gfCNCPoint1[6054] = {X 351.3681, Y 35.6206, Z -1.3333, A 0.000, B 0.000, C 0.000 }
gfCNCPoint1[6055] = {X 352.4747, Y 34.8217, Z -1.3333, A 0.000, B 0.000, C 0.000 }
gfCNCPoint1[6056] = {X 353.5730, Y 33.7520, Z -1.3333, A 0.000, B 0.000, C 0.000 }
gfCNCPoint1[6057] = {X 354.5237, Y 32.5493, Z -1.3333, A 0.000, B 0.000, C 0.000 }
gfCNCPoint1[6058] = {X 355.3108, Y 31.2336, Z -1.3333, A 0.000, B 0.000, C 0.000 }
gfCNCPoint1[6059] = {X 355.9209, Y 29.8271, Z -1.3333, A 0.000, B 0.000, C 0.000 }
gfCNCPoint1[6060] = {X 356.3440, Y 28.3535, Z -1.3333, A 0.000, B 0.000, C 0.000 }
gfCNCPoint1[6061] = {X 356.6085, Y 26.7184, Z -1.3333, A 0.000, B 0.000, C 0.000 }
gfCNCPoint1[6062] = {X 356.7162, Y 25.0656, Z -1.3333, A 0.000, B 0.000, C 0.000 }
gfCNCPoint1[6063] = {X 356.6661, Y 23.4100, Z -1.3333, A 0.000, B 0.000, C 0.000 }
gfCNCPoint1[6064] = {X 356.4586, Y 21.7667, Z -1.3333, A 0.000, B 0.000, C 0.000 }
gfCNCPoint1[6065] = {X 356.1382, Y 20.3836, Z -1.3333, A 0.000, B 0.000, C 0.000 }
gfCNCPoint1[6066] = {X 355.6490, Y 19.0509, Z -1.3333, A 0.000, B 0.000, C 0.000 }
gfCNCPoint1[6067] = {X 354.9985, Y 17.7891, Z -1.3333, A 0.000, B 0.000, C 0.000 }
gfCNCPoint1[6068] = {X 354.1969, Y 16.6174, Z -1.3333, A 0.000, B 0.000, C 0.000 }
gfCNCPoint1[6069] = {X 353.3646, Y 15.6889, Z -1.3333, A 0.000, B 0.000, C 0.000 }
gfCNCPoint1[6070] = {X 352.4079, Y 14.8891, Z -1.3333, A 0.000, B 0.000, C 0.000 }
gfCNCPoint1[6071] = {X 351.3465, Y 14.2346, Z -1.3333, A 0.000, B 0.000, C 0.000 }
gfCNCPoint1[6072] = {X 350.2023, Y 13.7390, Z -1.3333, A 0.000, B 0.000, C 0.000 }
gfCNCPoint1[6073] = {X 348.9989, Y 13.4124, Z -1.3333, A 0.000, B 0.000, C 0.000 }
gfCNCPoint1[6074] = {X 347.3616, Y 13.2058, Z -1.3333, A 0.000, B 0.000, C 0.000 }
gfCNCPoint1[6075] = {X 345.7114, Y 13.2112, Z -1.3333, A 0.000, B 0.000, C 0.000 }
gfCNCPoint1[6076] = {X 344.0755, Y 13.4284, Z -1.3333, A 0.000, B 0.000, C 0.000 }
gfCNCPoint1[6077] = {X 342.4811, Y 13.8538, Z -1.3333, A 0.000, B 0.000, C 0.000 }
gfCNCPoint1[6078] = {X 340.9545, Y 14.4805, Z -1.3333, A 0.000, B 0.000, C 0.000 }
gfCNCPoint1[6079] = {X 339.5210, Y 15.2981, Z -1.3333, A 0.000, B 0.000, C 0.000 }
gfCNCPoint1[6080] = {X 339.4274, Y 16.1841, Z -1.3333, A 0.000, B 0.000, C 0.000 }
gfCNCPoint1[6081] = {X 339.1743, Y 17.0384, Z -1.3333, A 0.000, B 0.000, C 0.000 }
gfCNCPoint1[6082] = {X 338.7701, Y 17.8324, Z -1.3333, A 0.000, B 0.000, C 0.000 }
gfCNCPoint1[6083] = {X 338.2283, Y 18.5396, Z -1.3333, A 0.000, B 0.000, C 0.000 }
gfCNCPoint1[6084] = {X 337.5670, Y 19.1366, Z -1.3333, A 0.000, B 0.000, C 0.000 }
gfCNCPoint1[6085] = {X 336.8399, Y 19.6716, Z -1.3333, A 0.000, B 0.000, C 0.000 }
gfCNCPoint1[6086] = {X 335.9170, Y 20.1909, Z -1.3333, A 0.000, B 0.000, C 0.000 }
gfCNCPoint1[6087] = {X 334.9039, Y 20.4988, Z -1.3333, A 0.000, B 0.000, C 0.000 }
gfCNCPoint1[6088] = {X 333.8481, Y 20.5809, Z -1.3333, A 0.000, B 0.000, C 0.000 }
gfCNCPoint1[6089] = {X 332.7995, Y 20.4334, Z -1.3333, A 0.000, B 0.000, C 0.000 }
gfCNCPoint1[6090] = {X 331.8074, Y 20.0631, Z -1.3333, A 0.000, B 0.000, C 0.000 }
gfCNCPoint1[6091] = {X 330.9185, Y 19.4875, Z -1.3333, A 0.000, B 0.000, C 0.000 }
gfCNCPoint1[6092] = {X 330.1748, Y 18.7338, Z -1.3333, A 0.000, B 0.000, C 0.000 }
gfCNCPoint1[6093] = {X 329.6111, Y 17.8373, Z -1.3333, A 0.000, B 0.000, C 0.000 }
gfCNCPoint1[6094] = {X 326.0906, Y 10.5950, Z -1.3333, A 0.000, B 0.000, C 0.000 }
gfCNCPoint1[6095] = {X 325.7555, Y 9.6856, Z -1.3333, A 0.000, B 0.000, C 0.000 }
gfCNCPoint1[6096] = {X 325.6068, Y 8.7279, Z -1.3333, A 0.000, B 0.000, C 0.000 }
gfCNCPoint1[6097] = {X 325.6502, Y 7.7597, Z -1.3333, A 0.000, B 0.000, C 0.000 }
gfCNCPoint1[6098] = {X 325.8841, Y 6.8192, Z -1.3333, A 0.000, B 0.000, C 0.000 }
gfCNCPoint1[6099] = {X 326.2993, Y 5.9435, Z -1.3333, A 0.000, B 0.000, C 0.000 }
gfCNCPoint1[6100] = {X 326.9295, Y 5.1131, Z -1.3333, A 0.000, B 0.000, C 0.000 }
gfCNCPoint1[6101] = {X 327.7216, Y 4.4356, Z -1.3333, A 0.000, B 0.000, C 0.000 }
gfCNCPoint1[6102] = {X 328.3967, Y 3.9733, Z -1.3333, A 0.000, B 0.000, C 0.000 }
gfCNCPoint1[6103] = {X 329.3298, Y 3.4827, Z -1.3333, A 0.000, B 0.000, C 0.000 }
gfCNCPoint1[6104] = {X 330.3464, Y 3.2039, Z -1.3333, A 0.000, B 0.000, C 0.000 }
gfCNCPoint1[6105] = {X 331.3992, Y 3.1499, Z -1.3333, A 0.000, B 0.000, C 0.000 }
gfCNCPoint1[6106] = {X 332.4390, Y 3.3233, Z -1.3333, A 0.000, B 0.000, C 0.000 }
gfCNCPoint1[6107] = {X 333.3767, Y 2.7966, Z -1.3333, A 0.000, B 0.000, C 0.000 }
gfCNCPoint1[6108] = {X 334.3334, Y 2.3051, Z -1.3333, A 0.000, B 0.000, C 0.000 }
gfCNCPoint1[6109] = {X 334.5448, Y 2.7361, Z -1.3333, A 0.000, B 0.000, C 0.000 }
gfCNCPoint1[6110] = {X 335.0204, Y 2.5083, Z -1.3333, A 0.000, B 0.000, C 0.000 }
gfCNCPoint1[6111] = {X 335.5002, Y 2.2893, Z -1.3333, A 0.000, B 0.000, C 0.000 }
gfCNCPoint1[6112] = {X 335.8480, Y 2.1345, Z -1.3333, A 0.000, B 0.000, C 0.000 }
gfCNCPoint1[6113] = {X 337.9511, Y 1.3140, Z -1.3333, A 0.000, B 0.000, C 0.000 }
gfCNCPoint1[6114] = {X 340.1167, Y 0.6764, Z -1.3333, A 0.000, B 0.000, C 0.000 }
gfCNCPoint1[6115] = {X 342.3290, Y 0.2265, Z -1.3333, A 0.000, B 0.000, C 0.000 }
gfCNCPoint1[6116] = {X 344.5716, Y -0.0325, Z -1.3333, A 0.000, B 0.000, C 0.000 }
gfCNCPoint1[6117] = {X 346.8281, Y -0.0986, Z -1.3333, A 0.000, B 0.000, C 0.000 }
gfCNCPoint1[6118] = {X 349.0821, Y 0.0286, Z -1.3333, A 0.000, B 0.000, C 0.000 }
gfCNCPoint1[6119] = {X 351.3169, Y 0.3481, Z -1.3333, A 0.000, B 0.000, C 0.000 }
gfCNCPoint1[6120] = {X 351.8868, Y 0.4533, Z -1.3333, A 0.000, B 0.000, C 0.000 }
gfCNCPoint1[6121] = {X 353.8281, Y 0.9413, Z -1.3333, A 0.000, B 0.000, C 0.000 }
gfCNCPoint1[6122] = {X 355.7145, Y 1.6111, Z -1.3333, A 0.000, B 0.000, C 0.000 }
gfCNCPoint1[6123] = {X 357.5290, Y 2.4565, Z -1.3333, A 0.000, B 0.000, C 0.000 }
gfCNCPoint1[6124] = {X 359.2553, Y 3.4699, Z -1.3333, A 0.000, B 0.000, C 0.000 }
gfCNCPoint1[6125] = {X 360.8778, Y 4.6423, Z -1.3333, A 0.000, B 0.000, C 0.000 }
gfCNCPoint1[6126] = {X 362.3820, Y 5.9632, Z -1.3333, A 0.000, B 0.000, C 0.000 }
gfCNCPoint1[6127] = {X 363.7542, Y 7.4205, Z -1.3333, A 0.000, B 0.000, C 0.000 }
gfCNCPoint1[6128] = {X 365.2289, Y 9.3236, Z -1.3333, A 0.000, B 0.000, C 0.000 }
gfCNCPoint1[6129] = {X 366.5120, Y 11.3606, Z -1.3333, A 0.000, B 0.000, C 0.000 }
gfCNCPoint1[6130] = {X 367.5917, Y 13.5125, Z -1.3333, A 0.000, B 0.000, C 0.000 }
gfCNCPoint1[6131] = {X 368.4575, Y 15.7589, Z -1.3333, A 0.000, B 0.000, C 0.000 }
gfCNCPoint1[6132] = {X 369.1015, Y 18.0787, Z -1.3333, A 0.000, B 0.000, C 0.000 }
gfCNCPoint1[6133] = {X 369.5814, Y 20.7163, Z -1.3333, A 0.000, B 0.000, C 0.000 }
gfCNCPoint1[6134] = {X 369.8368, Y 23.3851, Z -1.3333, A 0.000, B 0.000, C 0.000 }
gfCNCPoint1[6135] = {X 369.8659, Y 26.0659, Z -1.3333, A 0.000, B 0.000, C 0.000 }
gfCNCPoint1[6136] = {X 369.6685, Y 28.7395, Z -1.3333, A 0.000, B 0.000, C 0.000 }
gfCNCPoint1[6137] = {X 369.2461, Y 31.3870, Z -1.3333, A 0.000, B 0.000, C 0.000 }
gfCNCPoint1[6138] = {X 368.7206, Y 33.4984, Z -1.3333, A 0.000, B 0.000, C 0.000 }
gfCNCPoint1[6139] = {X 368.0105, Y 35.5551, Z -1.3333, A 0.000, B 0.000, C 0.000 }
gfCNCPoint1[6140] = {X 367.1214, Y 37.5409, Z -1.3333, A 0.000, B 0.000, C 0.000 }
gfCNCPoint1[6141] = {X 366.0603, Y 39.4405, Z -1.3333, A 0.000, B 0.000, C 0.000 }
gfCNCPoint1[6142] = {X 364.8354, Y 41.2387, Z -1.3333, A 0.000, B 0.000, C 0.000 }
gfCNCPoint1[6143] = {X 363.6033, Y 42.7570, Z -1.3333, A 0.000, B 0.000, C 0.000 }
gfCNCPoint1[6144] = {X 362.2428, Y 44.1612, Z -1.3333, A 0.000, B 0.000, C 0.000 }
gfCNCPoint1[6145] = {X 360.7642, Y 45.4407, Z -1.3333, A 0.000, B 0.000, C 0.000 }
gfCNCPoint1[6146] = {X 359.1791, Y 46.5854, Z -1.3333, A 0.000, B 0.000, C 0.000 }
gfCNCPoint1[6147] = {X 357.4997, Y 47.5867, Z -1.3333, A 0.000, B 0.000, C 0.000 }
gfCNCPoint1[6148] = {X 355.5329, Y 48.4795, Z -1.3333, A 0.000, B 0.000, C 0.000 }
gfCNCPoint1[6149] = {X 353.4902, Y 49.1814, Z -1.3333, A 0.000, B 0.000, C 0.000 }
gfCNCPoint1[6150] = {X 351.3901, Y 49.6861, Z -1.3333, A 0.000, B 0.000, C 0.000 }
gfCNCPoint1[6151] = {X 349.2515, Y 49.9891, Z -1.3333, A 0.000, B 0.000, C 0.000 }
gfCNCPoint1[6152] = {X 347.0938, Y 50.0876, Z -1.3333, A 0.000, B 0.000, C 0.000 }
gfCNCPoint1[6153] = {X 345.0197, Y 50.0525, Z -1.3333, A 0.000, B 0.000, C 0.000 }
gfCNCPoint1[6154] = {X 342.9564, Y 49.8375, Z -1.3333, A 0.000, B 0.000, C 0.000 }
gfCNCPoint1[6155] = {X 340.9196, Y 49.4444, Z -1.3333, A 0.000, B 0.000, C 0.000 }
gfCNCPoint1[6156] = {X 338.9245, Y 48.8760, Z -1.3333, A 0.000, B 0.000, C 0.000 }
gfCNCPoint1[6157] = {X 336.9863, Y 48.1366, Z -1.3333, A 0.000, B 0.000, C 0.000 }
gfCNCPoint1[6158] = {X 335.1196, Y 47.2319, Z -1.3333, A 0.000, B 0.000, C 0.000 }
gfCNCPoint1[6159] = {X 333.5425, Y 46.2572, Z -1.3333, A 0.000, B 0.000, C 0.000 }
gfCNCPoint1[6160] = {X 332.0447, Y 45.1645, Z -1.3333, A 0.000, B 0.000, C 0.000 }
gfCNCPoint1[6161] = {X 330.6350, Y 43.9603, Z -1.3333, A 0.000, B 0.000, C 0.000 }
gfCNCPoint1[6162] = {X 329.6763, Y 43.9518, Z -1.3333, A 0.000, B 0.000, C 0.000 }
gfCNCPoint1[6163] = {X 328.7422, Y 43.7359, Z -1.3333, A 0.000, B 0.000, C 0.000 }
gfCNCPoint1[6164] = {X 327.8771, Y 43.3228, Z -1.3333, A 0.000, B 0.000, C 0.000 }
gfCNCPoint1[6165] = {X 327.1219, Y 42.7321, Z -1.3333, A 0.000, B 0.000, C 0.000 }
gfCNCPoint1[6166] = {X 326.5249, Y 42.1498, Z -1.3333, A 0.000, B 0.000, C 0.000 }
gfCNCPoint1[6167] = {X 325.8848, Y 41.3619, Z -1.3333, A 0.000, B 0.000, C 0.000 }
gfCNCPoint1[6168] = {X 325.4424, Y 40.4483, Z -1.3333, A 0.000, B 0.000, C 0.000 }
gfCNCPoint1[6169] = {X 325.2210, Y 39.4576, Z -1.3333, A 0.000, B 0.000, C 0.000 }
gfCNCPoint1[6170] = {X 325.2326, Y 38.4426, Z -1.3333, A 0.000, B 0.000, C 0.000 }
gfCNCPoint1[6171] = {X 325.4765, Y 37.4572, Z -1.3333, A 0.000, B 0.000, C 0.000 }
gfCNCPoint1[6172] = {X 325.9397, Y 36.5539, Z -1.3333, A 0.000, B 0.000, C 0.000 }
gfCNCPoint1[6173] = {X 330.1988, Y 30.1861, Z -1.3333, A 0.000, B 0.000, C 0.000 }
gfCNCPoint1[6174] = {X 330.8195, Y 29.4619, Z -1.3333, A 0.000, B 0.000, C 0.000 }
gfCNCPoint1[6175] = {X 331.5817, Y 28.8884, Z -1.3333, A 0.000, B 0.000, C 0.000 }
gfCNCPoint1[6176] = {X 332.4495, Y 28.4927, Z -1.3333, A 0.000, B 0.000, C 0.000 }
gfCNCPoint1[6177] = {X 333.3822, Y 28.2932, Z -1.3333, A 0.000, B 0.000, C 0.000 }
gfCNCPoint1[6178] = {X 334.3360, Y 28.2995, Z -1.3333, A 0.000, B 0.000, C 0.000 }
gfCNCPoint1[6179] = {X 335.2660, Y 28.5111, Z -1.3333, A 0.000, B 0.000, C 0.000 }
gfCNCPoint1[6180] = {X 336.1286, Y 28.9182, Z -1.3333, A 0.000, B 0.000, C 0.000 }
gfCNCPoint1[6181] = {X 336.8832, Y 29.5016, Z -1.3333, A 0.000, B 0.000, C 0.000 }
gfCNCPoint1[6182] = {X 337.4845, Y 30.0811, Z -1.3333, A 0.000, B 0.000, C 0.000 }
gfCNCPoint1[6183] = {X 338.1274, Y 30.8804, Z -1.3333, A 0.000, B 0.000, C 0.000 }
gfCNCPoint1[6184] = {X 338.5678, Y 31.8068, Z -1.3333, A 0.000, B 0.000, C 0.000 }
gfCNCPoint1[6185] = {X 338.7817, Y 32.8100, Z -1.3333, A 0.000, B 0.000, C 0.000 }
gfCNCPoint1[6186] = {X 338.7575, Y 33.8355, Z -1.3333, A 0.000, B 0.000, C 0.000 }
gfCNCPoint1[6187] = {X 339.5029, Y 34.5092, Z -1.3333, A 0.000, B 0.000, C 0.000 }
gfCNCPoint1[6188] = {X 340.2812, Y 35.1446, Z -1.3333, A 0.000, B 0.000, C 0.000 }
gfCNCPoint1[6189] = {X 341.4925, Y 35.9471, Z -1.3333, A 0.000, B 0.000, C 0.000 }
gfCNCPoint1[6190] = {X 342.8028, Y 36.5754, Z -1.3333, A 0.000, B 0.000, C 0.000 }
gfCNCPoint1[6191] = {X 344.1871, Y 37.0173, Z -1.3333, A 0.000, B 0.000, C 0.000 }
gfCNCPoint1[6192] = {X 345.6190, Y 37.2646, Z -1.3333, A 0.000, B 0.000, C 0.000 }
gfCNCPoint1[6193] = {X 347.0713, Y 37.3125, Z -1.3333, A 0.000, B 0.000, C 0.000 }
gfCNCPoint1[6194] = {X 347.5133, Y 37.2896, Z -1.3333, A 0.000, B 0.000, C 0.000 }
gfCNCPoint1[6195] = {X 348.9438, Y 37.0973, Z -1.3333, A 0.000, B 0.000, C 0.000 }
gfCNCPoint1[6196] = {X 350.3238, Y 36.6741, Z -1.3333, A 0.000, B 0.000, C 0.000 }
gfCNCPoint1[6197] = {X 351.6163, Y 36.0314, Z -1.3333, A 0.000, B 0.000, C 0.000 }
gfCNCPoint1[6198] = {X 352.7866, Y 35.1865, Z -1.3333, A 0.000, B 0.000, C 0.000 }
gfCNCPoint1[6199] = {X 353.9297, Y 34.0732, Z -1.3333, A 0.000, B 0.000, C 0.000 }
gfCNCPoint1[6200] = {X 354.9191, Y 32.8214, Z -1.3333, A 0.000, B 0.000, C 0.000 }
gfCNCPoint1[6201] = {X 355.7382, Y 31.4519, Z -1.3333, A 0.000, B 0.000, C 0.000 }
gfCNCPoint1[6202] = {X 356.3731, Y 29.9880, Z -1.3333, A 0.000, B 0.000, C 0.000 }
gfCNCPoint1[6203] = {X 356.8133, Y 28.4543, Z -1.3333, A 0.000, B 0.000, C 0.000 }
gfCNCPoint1[6204] = {X 357.0854, Y 26.7729, Z -1.3333, A 0.000, B 0.000, C 0.000 }
gfCNCPoint1[6205] = {X 357.1961, Y 25.0733, Z -1.3333, A 0.000, B 0.000, C 0.000 }
gfCNCPoint1[6206] = {X 357.1445, Y 23.3709, Z -1.3333, A 0.000, B 0.000, C 0.000 }
gfCNCPoint1[6207] = {X 356.9309, Y 21.6811, Z -1.3333, A 0.000, B 0.000, C 0.000 }
gfCNCPoint1[6208] = {X 356.5967, Y 20.2416, Z -1.3333, A 0.000, B 0.000, C 0.000 }
gfCNCPoint1[6209] = {X 356.0869, Y 18.8544, Z -1.3333, A 0.000, B 0.000, C 0.000 }
gfCNCPoint1[6210] = {X 355.4094, Y 17.5410, Z -1.3333, A 0.000, B 0.000, C 0.000 }
gfCNCPoint1[6211] = {X 354.5747, Y 16.3214, Z -1.3333, A 0.000, B 0.000, C 0.000 }
gfCNCPoint1[6212] = {X 353.6964, Y 15.3420, Z -1.3333, A 0.000, B 0.000, C 0.000 }
gfCNCPoint1[6213] = {X 352.6869, Y 14.4985, Z -1.3333, A 0.000, B 0.000, C 0.000 }
gfCNCPoint1[6214] = {X 351.5670, Y 13.8083, Z -1.3333, A 0.000, B 0.000, C 0.000 }
gfCNCPoint1[6215] = {X 350.3598, Y 13.2856, Z -1.3333, A 0.000, B 0.000, C 0.000 }
gfCNCPoint1[6216] = {X 349.0902, Y 12.9412, Z -1.3333, A 0.000, B 0.000, C 0.000 }
gfCNCPoint1[6217] = {X 347.3476, Y 12.7241, Z -1.3333, A 0.000, B 0.000, C 0.000 }
gfCNCPoint1[6218] = {X 345.5915, Y 12.7385, Z -1.3333, A 0.000, B 0.000, C 0.000 }
gfCNCPoint1[6219] = {X 343.8527, Y 12.9840, Z -1.3333, A 0.000, B 0.000, C 0.000 }
gfCNCPoint1[6220] = {X 342.1613, Y 13.4563, Z -1.3333, A 0.000, B 0.000, C 0.000 }
gfCNCPoint1[6221] = {X 340.5469, Y 14.1474, Z -1.3333, A 0.000, B 0.000, C 0.000 }
gfCNCPoint1[6222] = {X 339.0375, Y 15.0450, Z -1.3333, A 0.000, B 0.000, C 0.000 }
gfCNCPoint1[6223] = {X 338.9897, Y 15.9032, Z -1.3333, A 0.000, B 0.000, C 0.000 }
gfCNCPoint1[6224] = {X 338.7760, Y 16.7358, Z -1.3333, A 0.000, B 0.000, C 0.000 }
gfCNCPoint1[6225] = {X 338.4045, Y 17.5109, Z -1.3333, A 0.000, B 0.000, C 0.000 }
gfCNCPoint1[6226] = {X 337.8894, Y 18.1990, Z -1.3333, A 0.000, B 0.000, C 0.000 }
gfCNCPoint1[6227] = {X 337.2504, Y 18.7738, Z -1.3333, A 0.000, B 0.000, C 0.000 }
gfCNCPoint1[6228] = {X 336.5606, Y 19.2813, Z -1.3333, A 0.000, B 0.000, C 0.000 }
gfCNCPoint1[6229] = {X 335.7284, Y 19.7495, Z -1.3333, A 0.000, B 0.000, C 0.000 }
gfCNCPoint1[6230] = {X 334.8148, Y 20.0271, Z -1.3333, A 0.000, B 0.000, C 0.000 }
gfCNCPoint1[6231] = {X 333.8628, Y 20.1012, Z -1.3333, A 0.000, B 0.000, C 0.000 }
gfCNCPoint1[6232] = {X 332.9173, Y 19.9681, Z -1.3333, A 0.000, B 0.000, C 0.000 }
gfCNCPoint1[6233] = {X 332.0228, Y 19.6341, Z -1.3333, A 0.000, B 0.000, C 0.000 }
gfCNCPoint1[6234] = {X 331.2213, Y 19.1151, Z -1.3333, A 0.000, B 0.000, C 0.000 }
gfCNCPoint1[6235] = {X 330.5507, Y 18.4353, Z -1.3333, A 0.000, B 0.000, C 0.000 }
gfCNCPoint1[6236] = {X 330.0425, Y 17.6269, Z -1.3333, A 0.000, B 0.000, C 0.000 }
gfCNCPoint1[6237] = {X 326.5223, Y 10.3852, Z -1.3333, A 0.000, B 0.000, C 0.000 }
gfCNCPoint1[6238] = {X 326.2154, Y 9.5469, Z -1.3333, A 0.000, B 0.000, C 0.000 }
gfCNCPoint1[6239] = {X 326.0841, Y 8.6639, Z -1.3333, A 0.000, B 0.000, C 0.000 }
gfCNCPoint1[6240] = {X 326.1338, Y 7.7725, Z -1.3333, A 0.000, B 0.000, C 0.000 }
gfCNCPoint1[6241] = {X 326.3623, Y 6.9096, Z -1.3333, A 0.000, B 0.000, C 0.000 }
gfCNCPoint1[6242] = {X 326.7603, Y 6.1105, Z -1.3333, A 0.000, B 0.000, C 0.000 }
gfCNCPoint1[6243] = {X 327.3114, Y 5.4082, Z -1.3333, A 0.000, B 0.000, C 0.000 }
gfCNCPoint1[6244] = {X 327.9929, Y 4.8316, Z -1.3333, A 0.000, B 0.000, C 0.000 }
gfCNCPoint1[6245] = {X 328.6647, Y 4.3715, Z -1.3333, A 0.000, B 0.000, C 0.000 }
gfCNCPoint1[6246] = {X 329.5528, Y 3.9110, Z -1.3333, A 0.000, B 0.000, C 0.000 }
gfCNCPoint1[6247] = {X 330.5219, Y 3.6630, Z -1.3333, A 0.000, B 0.000, C 0.000 }
gfCNCPoint1[6248] = {X 331.5220, Y 3.6403, Z -1.3333, A 0.000, B 0.000, C 0.000 }
gfCNCPoint1[6249] = {X 332.5013, Y 3.8441, Z -1.3333, A 0.000, B 0.000, C 0.000 }
gfCNCPoint1[6250] = {X 333.5117, Y 3.2692, Z -1.3333, A 0.000, B 0.000, C 0.000 }
gfCNCPoint1[6251] = {X 334.5448, Y 2.7361, Z -1.3333, A 0.000, B 0.000, C 0.000 }
gfCNCPoint1[6252] = {X 334.3334, Y 2.3051, Z -1.3333, A 0.000, B 0.000, C 0.000 }
gfCNCPoint1[6253] = {X 2.3035, Y 2.3051, Z -1.3333, A 0.000, B 0.000, C 0.000 }
gfCNCPoint1[6254] = {X 2.3035, Y 6.8598, Z -1.3333, A 0.000, B 0.000, C 0.000 }
gfCNCPoint1[6255] = {X 2.4148, Y 6.8820, Z -1.3333, A 0.000, B 0.000, C 0.000 }
gfCNCPoint1[6256] = {X 2.8633, Y 6.6974, Z -1.3333, A 0.000, B 0.000, C 0.000 }
gfCNCPoint1[6257] = {X 3.3170, Y 6.5258, Z -1.3333, A 0.000, B 0.000, C 0.000 }
gfCNCPoint1[6258] = {X 5.4241, Y 5.7921, Z -1.3333, A 0.000, B 0.000, C 0.000 }
gfCNCPoint1[6259] = {X 7.5864, Y 5.2420, Z -1.3333, A 0.000, B 0.000, C 0.000 }
gfCNCPoint1[6260] = {X 9.7880, Y 4.8799, Z -1.3333, A 0.000, B 0.000, C 0.000 }
gfCNCPoint1[6261] = {X 12.0125, Y 4.7083, Z -1.3333, A 0.000, B 0.000, C 0.000 }
gfCNCPoint1[6262] = {X 14.2436, Y 4.7284, Z -1.3333, A 0.000, B 0.000, C 0.000 }
gfCNCPoint1[6263] = {X 16.4647, Y 4.9402, Z -1.3333, A 0.000, B 0.000, C 0.000 }
gfCNCPoint1[6264] = {X 18.0939, Y 5.2209, Z -1.3333, A 0.000, B 0.000, C 0.000 }
gfCNCPoint1[6265] = {X 19.6943, Y 5.6356, Z -1.3333, A 0.000, B 0.000, C 0.000 }
gfCNCPoint1[6266] = {X 21.2549, Y 6.1815, Z -1.3333, A 0.000, B 0.000, C 0.000 }
gfCNCPoint1[6267] = {X 22.7648, Y 6.8547, Z -1.3333, A 0.000, B 0.000, C 0.000 }
gfCNCPoint1[6268] = {X 24.4874, Y 7.8191, Z -1.3333, A 0.000, B 0.000, C 0.000 }
gfCNCPoint1[6269] = {X 26.1061, Y 8.9491, Z -1.3333, A 0.000, B 0.000, C 0.000 }
gfCNCPoint1[6270] = {X 27.3994, Y 10.0793, Z -1.3333, A 0.000, B 0.000, C 0.000 }
gfCNCPoint1[6271] = {X 28.5597, Y 11.3458, Z -1.3333, A 0.000, B 0.000, C 0.000 }
gfCNCPoint1[6272] = {X 29.5727, Y 12.7328, Z -1.3333, A 0.000, B 0.000, C 0.000 }
gfCNCPoint1[6273] = {X 30.4260, Y 14.2235, Z -1.3333, A 0.000, B 0.000, C 0.000 }
gfCNCPoint1[6274] = {X 31.1090, Y 15.7994, Z -1.3333, A 0.000, B 0.000, C 0.000 }
gfCNCPoint1[6275] = {X 31.6681, Y 17.7351, Z -1.3333, A 0.000, B 0.000, C 0.000 }
gfCNCPoint1[6276] = {X 32.0010, Y 19.7223, Z -1.3333, A 0.000, B 0.000, C 0.000 }
gfCNCPoint1[6277] = {X 32.1035, Y 21.7345, Z -1.3333, A 0.000, B 0.000, C 0.000 }
gfCNCPoint1[6278] = {X 31.9740, Y 23.7452, Z -1.3333, A 0.000, B 0.000, C 0.000 }
gfCNCPoint1[6279] = {X 31.6144, Y 25.7277, Z -1.3333, A 0.000, B 0.000, C 0.000 }
gfCNCPoint1[6280] = {X 31.1957, Y 27.1568, Z -1.3333, A 0.000, B 0.000, C 0.000 }
gfCNCPoint1[6281] = {X 30.6294, Y 28.5341, Z -1.3333, A 0.000, B 0.000, C 0.000 }
gfCNCPoint1[6282] = {X 29.9217, Y 29.8443, Z -1.3333, A 0.000, B 0.000, C 0.000 }
gfCNCPoint1[6283] = {X 29.0802, Y 31.0729, Z -1.3333, A 0.000, B 0.000, C 0.000 }
gfCNCPoint1[6284] = {X 29.6384, Y 31.7917, Z -1.3333, A 0.000, B 0.000, C 0.000 }
gfCNCPoint1[6285] = {X 30.0955, Y 32.5786, Z -1.3333, A 0.000, B 0.000, C 0.000 }
gfCNCPoint1[6286] = {X 33.1423, Y 38.8726, Z -1.3333, A 0.000, B 0.000, C 0.000 }
gfCNCPoint1[6287] = {X 33.5391, Y 39.8957, Z -1.3333, A 0.000, B 0.000, C 0.000 }
gfCNCPoint1[6288] = {X 33.7662, Y 40.9694, Z -1.3333, A 0.000, B 0.000, C 0.000 }
gfCNCPoint1[6289] = {X 33.8177, Y 42.0656, Z -1.3333, A 0.000, B 0.000, C 0.000 }
gfCNCPoint1[6290] = {X 33.7164, Y 43.0266, Z -1.3333, A 0.000, B 0.000, C 0.000 }
gfCNCPoint1[6291] = {X 33.4799, Y 43.9636, Z -1.3333, A 0.000, B 0.000, C 0.000 }
gfCNCPoint1[6292] = {X 33.1103, Y 44.8630, Z -1.3333, A 0.000, B 0.000, C 0.000 }
gfCNCPoint1[6293] = {X 32.6161, Y 45.7005, Z -1.3333, A 0.000, B 0.000, C 0.000 }
gfCNCPoint1[6294] = {X 32.0075, Y 46.4590, Z -1.3333, A 0.000, B 0.000, C 0.000 }
gfCNCPoint1[6295] = {X 31.2970, Y 47.1229, Z -1.3333, A 0.000, B 0.000, C 0.000 }
gfCNCPoint1[6296] = {X 30.7576, Y 47.5591, Z -1.3333, A 0.000, B 0.000, C 0.000 }
gfCNCPoint1[6297] = {X 29.8516, Y 48.1761, Z -1.3333, A 0.000, B 0.000, C 0.000 }
gfCNCPoint1[6298] = {X 28.8585, Y 48.6400, Z -1.3333, A 0.000, B 0.000, C 0.000 }
gfCNCPoint1[6299] = {X 27.8039, Y 48.9388, Z -1.3333, A 0.000, B 0.000, C 0.000 }
gfCNCPoint1[6300] = {X 26.7150, Y 49.0648, Z -1.3333, A 0.000, B 0.000, C 0.000 }
gfCNCPoint1[6301] = {X 25.6200, Y 49.0146, Z -1.3333, A 0.000, B 0.000, C 0.000 }
gfCNCPoint1[6302] = {X 23.6827, Y 49.9677, Z -1.3333, A 0.000, B 0.000, C 0.000 }
gfCNCPoint1[6303] = {X 21.6835, Y 50.7833, Z -1.3333, A 0.000, B 0.000, C 0.000 }
gfCNCPoint1[6304] = {X 19.6323, Y 51.4573, Z -1.3333, A 0.000, B 0.000, C 0.000 }
gfCNCPoint1[6305] = {X 19.1081, Y 51.6028, Z -1.3333, A 0.000, B 0.000, C 0.000 }
gfCNCPoint1[6306] = {X 17.0367, Y 52.0819, Z -1.3333, A 0.000, B 0.000, C 0.000 }
gfCNCPoint1[6307] = {X 14.9318, Y 52.3815, Z -1.3333, A 0.000, B 0.000, C 0.000 }
gfCNCPoint1[6308] = {X 12.8089, Y 52.4993, Z -1.3333, A 0.000, B 0.000, C 0.000 }
gfCNCPoint1[6309] = {X 10.6838, Y 52.4344, Z -1.3333, A 0.000, B 0.000, C 0.000 }
gfCNCPoint1[6310] = {X 8.5721, Y 52.1873, Z -1.3333, A 0.000, B 0.000, C 0.000 }
gfCNCPoint1[6311] = {X 6.9848, Y 51.8941, Z -1.3333, A 0.000, B 0.000, C 0.000 }
gfCNCPoint1[6312] = {X 5.4269, Y 51.4713, Z -1.3333, A 0.000, B 0.000, C 0.000 }
gfCNCPoint1[6313] = {X 3.8373, Y 50.8924, Z -1.3333, A 0.000, B 0.000, C 0.000 }
gfCNCPoint1[6314] = {X 2.3035, Y 50.1786, Z -1.3333, A 0.000, B 0.000, C 0.000 }
gfCNCPoint1[6315] = {X 2.3035, Y 97.6949, Z -1.3333, A 0.000, B 0.000, C 0.000 }
gfCNCPoint1[6316] = {X 120.1200, Y 97.6949, Z -1.3333, A 0.000, B 0.000, C 0.000 }
gfCNCPoint1[6317] = {X 120.1200, Y 97.0659, Z -1.3333, A 0.000, B 0.000, C 0.000 }
gfCNCPoint1[6318] = {X 120.2340, Y 96.0173, Z -1.3333, A 0.000, B 0.000, C 0.000 }
gfCNCPoint1[6319] = {X 120.5707, Y 95.0176, Z -1.3333, A 0.000, B 0.000, C 0.000 }
gfCNCPoint1[6320] = {X 121.1143, Y 94.1136, Z -1.3333, A 0.000, B 0.000, C 0.000 }
gfCNCPoint1[6321] = {X 121.8395, Y 93.3476, Z -1.3333, A 0.000, B 0.000, C 0.000 }
gfCNCPoint1[6322] = {X 122.7124, Y 92.7553, Z -1.3333, A 0.000, B 0.000, C 0.000 }
gfCNCPoint1[6323] = {X 123.6922, Y 92.3644, Z -1.3333, A 0.000, B 0.000, C 0.000 }
gfCNCPoint1[6324] = {X 124.7330, Y 92.1932, Z -1.3333, A 0.000, B 0.000, C 0.000 }
gfCNCPoint1[6325] = {X 124.7890, Y 92.1792, Z -1.3333, A 0.000, B 0.000, C 0.000 }
gfCNCPoint1[6326] = {X 124.8458, Y 92.1689, Z -1.3333, A 0.000, B 0.000, C 0.000 }
gfCNCPoint1[6327] = {X 125.3649, Y 92.0918, Z -1.3333, A 0.000, B 0.000, C 0.000 }
gfCNCPoint1[6328] = {X 126.1002, Y 91.9698, Z -1.3333, A 0.000, B 0.000, C 0.000 }
gfCNCPoint1[6329] = {X 126.8265, Y 91.8027, Z -1.3333, A 0.000, B 0.000, C 0.000 }
gfCNCPoint1[6330] = {X 127.9745, Y 90.7130, Z -1.3333, A 0.000, B 0.000, C 0.000 }
gfCNCPoint1[6331] = {X 129.0643, Y 89.5653, Z -1.3333, A 0.000, B 0.000, C 0.000 }
gfCNCPoint1[6332] = {X 154.9465, Y 61.1430, Z -1.3333, A 0.000, B 0.000, C 0.000 }
gfCNCPoint1[6333] = {X 154.6595, Y 60.4502, Z -1.3333, A 0.000, B 0.000, C 0.000 }
gfCNCPoint1[6334] = {X 154.4819, Y 59.7216, Z -1.3333, A 0.000, B 0.000, C 0.000 }
gfCNCPoint1[6335] = {X 154.4181, Y 58.9744, Z -1.3333, A 0.000, B 0.000, C 0.000 }
gfCNCPoint1[6336] = {X 154.4180, Y 58.0000, Z -1.3333, A 0.000, B 0.000, C 0.000 }
gfCNCPoint1[6337] = {X 154.5117, Y 57.0480, Z -1.3333, A 0.000, B 0.000, C 0.000 }
gfCNCPoint1[6338] = {X 154.7894, Y 56.1325, Z -1.3333, A 0.000, B 0.000, C 0.000 }
gfCNCPoint1[6339] = {X 155.2404, Y 55.2888, Z -1.3333, A 0.000, B 0.000, C 0.000 }
gfCNCPoint1[6340] = {X 155.8473, Y 54.5493, Z -1.3333, A 0.000, B 0.000, C 0.000 }
gfCNCPoint1[6341] = {X 156.5868, Y 53.9424, Z -1.3333, A 0.000, B 0.000, C 0.000 }
gfCNCPoint1[6342] = {X 157.4305, Y 53.4915, Z -1.3333, A 0.000, B 0.000, C 0.000 }
gfCNCPoint1[6343] = {X 158.3459, Y 53.2138, Z -1.3333, A 0.000, B 0.000, C 0.000 }
gfCNCPoint1[6344] = {X 159.2980, Y 53.1200, Z -1.3333, A 0.000, B 0.000, C 0.000 }
gfCNCPoint1[6345] = {X 178.5335, Y 53.1200, Z -1.3333, A 0.000, B 0.000, C 0.000 }
gfCNCPoint1[6346] = {X 179.4855, Y 53.2138, Z -1.3333, A 0.000, B 0.000, C 0.000 }
gfCNCPoint1[6347] = {X 180.4010, Y 53.4915, Z -1.3333, A 0.000, B 0.000, C 0.000 }
gfCNCPoint1[6348] = {X 181.2447, Y 53.9424, Z -1.3333, A 0.000, B 0.000, C 0.000 }
gfCNCPoint1[6349] = {X 181.9842, Y 54.5493, Z -1.3333, A 0.000, B 0.000, C 0.000 }
gfCNCPoint1[6350] = {X 182.5911, Y 55.2888, Z -1.3333, A 0.000, B 0.000, C 0.000 }
gfCNCPoint1[6351] = {X 183.0420, Y 56.1325, Z -1.3333, A 0.000, B 0.000, C 0.000 }
gfCNCPoint1[6352] = {X 183.3197, Y 57.0480, Z -1.3333, A 0.000, B 0.000, C 0.000 }
gfCNCPoint1[6353] = {X 183.4135, Y 58.0000, Z -1.3333, A 0.000, B 0.000, C 0.000 }
gfCNCPoint1[6354] = {X 183.4133, Y 58.9744, Z -1.3333, A 0.000, B 0.000, C 0.000 }
gfCNCPoint1[6355] = {X 183.3512, Y 59.7116, Z -1.3333, A 0.000, B 0.000, C 0.000 }
gfCNCPoint1[6356] = {X 183.1782, Y 60.4310, Z -1.3333, A 0.000, B 0.000, C 0.000 }
gfCNCPoint1[6357] = {X 182.8986, Y 61.1159, Z -1.3333, A 0.000, B 0.000, C 0.000 }
gfCNCPoint1[6358] = {X 209.8900, Y 90.5755, Z -1.3333, A 0.000, B 0.000, C 0.000 }
gfCNCPoint1[6359] = {X 210.5198, Y 91.2145, Z -1.3333, A 0.000, B 0.000, C 0.000 }
gfCNCPoint1[6360] = {X 211.1945, Y 91.8059, Z -1.3333, A 0.000, B 0.000, C 0.000 }
gfCNCPoint1[6361] = {X 211.3567, Y 91.9083, Z -1.3333, A 0.000, B 0.000, C 0.000 }
gfCNCPoint1[6362] = {X 211.5387, Y 91.9690, Z -1.3333, A 0.000, B 0.000, C 0.000 }
gfCNCPoint1[6363] = {X 212.4766, Y 92.1443, Z -1.3333, A 0.000, B 0.000, C 0.000 }
gfCNCPoint1[6364] = {X 213.4244, Y 92.2543, Z -1.3333, A 0.000, B 0.000, C 0.000 }
gfCNCPoint1[6365] = {X 214.4487, Y 92.1769, Z -1.3333, A 0.000, B 0.000, C 0.000 }
gfCNCPoint1[6366] = {X 215.4743, Y 92.1178, Z -1.3333, A 0.000, B 0.000, C 0.000 }
gfCNCPoint1[6367] = {X 216.0497, Y 92.0584, Z -1.3333, A 0.000, B 0.000, C 0.000 }
gfCNCPoint1[6368] = {X 216.6041, Y 91.8930, Z -1.3333, A 0.000, B 0.000, C 0.000 }
gfCNCPoint1[6369] = {X 217.1181, Y 91.6274, Z -1.3333, A 0.000, B 0.000, C 0.000 }
gfCNCPoint1[6370] = {X 244.6023, Y 74.0194, Z -1.3333, A 0.000, B 0.000, C 0.000 }
gfCNCPoint1[6371] = {X 221.4278, Y 64.9244, Z -1.3333, A 0.000, B 0.000, C 0.000 }
gfCNCPoint1[6372] = {X 219.7201, Y 64.3522, Z -1.3333, A 0.000, B 0.000, C 0.000 }
gfCNCPoint1[6373] = {X 217.9581, Y 63.9795, Z -1.3333, A 0.000, B 0.000, C 0.000 }
gfCNCPoint1[6374] = {X 216.1649, Y 63.8112, Z -1.3333, A 0.000, B 0.000, C 0.000 }
gfCNCPoint1[6375] = {X 215.1123, Y 63.6595, Z -1.3333, A 0.000, B 0.000, C 0.000 }
gfCNCPoint1[6376] = {X 214.1176, Y 63.2833, Z -1.3333, A 0.000, B 0.000, C 0.000 }
gfCNCPoint1[6377] = {X 213.2279, Y 62.7006, Z -1.3333, A 0.000, B 0.000, C 0.000 }
gfCNCPoint1[6378] = {X 212.4857, Y 61.9390, Z -1.3333, A 0.000, B 0.000, C 0.000 }
gfCNCPoint1[6379] = {X 211.9260, Y 61.0346, Z -1.3333, A 0.000, B 0.000, C 0.000 }
gfCNCPoint1[6380] = {X 211.5756, Y 60.0305, Z -1.3333, A 0.000, B 0.000, C 0.000 }
gfCNCPoint1[6381] = {X 211.4510, Y 58.9744, Z -1.3333, A 0.000, B 0.000, C 0.000 }
gfCNCPoint1[6382] = {X 211.4508, Y 58.0000, Z -1.3333, A 0.000, B 0.000, C 0.000 }
gfCNCPoint1[6383] = {X 211.5446, Y 57.0480, Z -1.3333, A 0.000, B 0.000, C 0.000 }
gfCNCPoint1[6384] = {X 211.8223, Y 56.1325, Z -1.3333, A 0.000, B 0.000, C 0.000 }
gfCNCPoint1[6385] = {X 212.2732, Y 55.2888, Z -1.3333, A 0.000, B 0.000, C 0.000 }
gfCNCPoint1[6386] = {X 212.8801, Y 54.5493, Z -1.3333, A 0.000, B 0.000, C 0.000 }
gfCNCPoint1[6387] = {X 213.6196, Y 53.9424, Z -1.3333, A 0.000, B 0.000, C 0.000 }
gfCNCPoint1[6388] = {X 214.4633, Y 53.4915, Z -1.3333, A 0.000, B 0.000, C 0.000 }
gfCNCPoint1[6389] = {X 215.3788, Y 53.2138, Z -1.3333, A 0.000, B 0.000, C 0.000 }
gfCNCPoint1[6390] = {X 216.3308, Y 53.1200, Z -1.3333, A 0.000, B 0.000, C 0.000 }
gfCNCPoint1[6391] = {X 237.2617, Y 53.1200, Z -1.3333, A 0.000, B 0.000, C 0.000 }
gfCNCPoint1[6392] = {X 238.3266, Y 53.2376, Z -1.3333, A 0.000, B 0.000, C 0.000 }
gfCNCPoint1[6393] = {X 239.3402, Y 53.5848, Z -1.3333, A 0.000, B 0.000, C 0.000 }
gfCNCPoint1[6394] = {X 240.2536, Y 54.1448, Z -1.3333, A 0.000, B 0.000, C 0.000 }
gfCNCPoint1[6395] = {X 241.0228, Y 54.8906, Z -1.3333, A 0.000, B 0.000, C 0.000 }
gfCNCPoint1[6396] = {X 241.6107, Y 55.7862, Z -1.3333, A 0.000, B 0.000, C 0.000 }
gfCNCPoint1[6397] = {X 241.9890, Y 56.7886, Z -1.3333, A 0.000, B 0.000, C 0.000 }
gfCNCPoint1[6398] = {X 242.1394, Y 57.8494, Z -1.3333, A 0.000, B 0.000, C 0.000 }
gfCNCPoint1[6399] = {X 248.3199, Y 60.2591, Z -1.3333, A 0.000, B 0.000, C 0.000 }
gfCNCPoint1[6400] = {X 275.0740, Y 70.8783, Z -1.3333, A 0.000, B 0.000, C 0.000 }
gfCNCPoint1[6401] = {X 275.0733, Y 63.6743, Z -1.3333, A 0.000, B 0.000, C 0.000 }
gfCNCPoint1[6402] = {X 274.0649, Y 63.3061, Z -1.3333, A 0.000, B 0.000, C 0.000 }
gfCNCPoint1[6403] = {X 273.1613, Y 62.7263, Z -1.3333, A 0.000, B 0.000, C 0.000 }
gfCNCPoint1[6404] = {X 272.4064, Y 61.9629, Z -1.3333, A 0.000, B 0.000, C 0.000 }
gfCNCPoint1[6405] = {X 271.8367, Y 61.0530, Z -1.3333, A 0.000, B 0.000, C 0.000 }
gfCNCPoint1[6406] = {X 271.4798, Y 60.0404, Z -1.3333, A 0.000, B 0.000, C 0.000 }
gfCNCPoint1[6407] = {X 271.3529, Y 58.9744, Z -1.3333, A 0.000, B 0.000, C 0.000 }
gfCNCPoint1[6408] = {X 271.3527, Y 58.0000, Z -1.3333, A 0.000, B 0.000, C 0.000 }
gfCNCPoint1[6409] = {X 271.4465, Y 57.0480, Z -1.3333, A 0.000, B 0.000, C 0.000 }
gfCNCPoint1[6410] = {X 271.7242, Y 56.1325, Z -1.3333, A 0.000, B 0.000, C 0.000 }
gfCNCPoint1[6411] = {X 272.1751, Y 55.2888, Z -1.3333, A 0.000, B 0.000, C 0.000 }
gfCNCPoint1[6412] = {X 272.7820, Y 54.5493, Z -1.3333, A 0.000, B 0.000, C 0.000 }
gfCNCPoint1[6413] = {X 273.5215, Y 53.9424, Z -1.3333, A 0.000, B 0.000, C 0.000 }
gfCNCPoint1[6414] = {X 274.3652, Y 53.4915, Z -1.3333, A 0.000, B 0.000, C 0.000 }
gfCNCPoint1[6415] = {X 275.2806, Y 53.2138, Z -1.3333, A 0.000, B 0.000, C 0.000 }
gfCNCPoint1[6416] = {X 276.2327, Y 53.1200, Z -1.3333, A 0.000, B 0.000, C 0.000 }
gfCNCPoint1[6417] = {X 292.7731, Y 53.1200, Z -1.3333, A 0.000, B 0.000, C 0.000 }
gfCNCPoint1[6418] = {X 293.7251, Y 53.2138, Z -1.3333, A 0.000, B 0.000, C 0.000 }
gfCNCPoint1[6419] = {X 294.6406, Y 53.4915, Z -1.3333, A 0.000, B 0.000, C 0.000 }
gfCNCPoint1[6420] = {X 295.4843, Y 53.9424, Z -1.3333, A 0.000, B 0.000, C 0.000 }
gfCNCPoint1[6421] = {X 296.2238, Y 54.5493, Z -1.3333, A 0.000, B 0.000, C 0.000 }
gfCNCPoint1[6422] = {X 296.8307, Y 55.2888, Z -1.3333, A 0.000, B 0.000, C 0.000 }
gfCNCPoint1[6423] = {X 297.2816, Y 56.1325, Z -1.3333, A 0.000, B 0.000, C 0.000 }
gfCNCPoint1[6424] = {X 297.5593, Y 57.0480, Z -1.3333, A 0.000, B 0.000, C 0.000 }
gfCNCPoint1[6425] = {X 297.6531, Y 58.0000, Z -1.3333, A 0.000, B 0.000, C 0.000 }
gfCNCPoint1[6426] = {X 297.6531, Y 58.9372, Z -1.3333, A 0.000, B 0.000, C 0.000 }
gfCNCPoint1[6427] = {X 297.5303, Y 60.0093, Z -1.3333, A 0.000, B 0.000, C 0.000 }
gfCNCPoint1[6428] = {X 297.1758, Y 61.0285, Z -1.3333, A 0.000, B 0.000, C 0.000 }
gfCNCPoint1[6429] = {X 296.6066, Y 61.9453, Z -1.3333, A 0.000, B 0.000, C 0.000 }
gfCNCPoint1[6430] = {X 295.8505, Y 62.7152, Z -1.3333, A 0.000, B 0.000, C 0.000 }
gfCNCPoint1[6431] = {X 294.9441, Y 63.3008, Z -1.3333, A 0.000, B 0.000, C 0.000 }
gfCNCPoint1[6432] = {X 293.9314, Y 63.6737, Z -1.3333, A 0.000, B 0.000, C 0.000 }
gfCNCPoint1[6433] = {X 293.9314, Y 92.3212, Z -1.3333, A 0.000, B 0.000, C 0.000 }
gfCNCPoint1[6434] = {X 294.9440, Y 92.6966, Z -1.3333, A 0.000, B 0.000, C 0.000 }
gfCNCPoint1[6435] = {X 295.8501, Y 93.2842, Z -1.3333, A 0.000, B 0.000, C 0.000 }
gfCNCPoint1[6436] = {X 296.6059, Y 94.0555, Z -1.3333, A 0.000, B 0.000, C 0.000 }
gfCNCPoint1[6437] = {X 297.1749, Y 94.9733, Z -1.3333, A 0.000, B 0.000, C 0.000 }
gfCNCPoint1[6438] = {X 297.5297, Y 95.9933, Z -1.3333, A 0.000, B 0.000, C 0.000 }
gfCNCPoint1[6439] = {X 297.6531, Y 97.0661, Z -1.3333, A 0.000, B 0.000, C 0.000 }
gfCNCPoint1[6440] = {X 297.6531, Y 97.6949, Z -1.3333, A 0.000, B 0.000, C 0.000 }
gfCNCPoint1[6441] = {X 297.1731, Y 97.6949, Z -1.3333, A 0.000, B 0.000, C 0.000 }
gfCNCPoint1[6442] = {X 297.1731, Y 98.0000, Z -1.3333, A 0.000, B 0.000, C 0.000 }
gfCNCPoint1[6443] = {X 297.0628, Y 98.9791, Z -1.3333, A 0.000, B 0.000, C 0.000 }
gfCNCPoint1[6444] = {X 296.7373, Y 99.9091, Z -1.3333, A 0.000, B 0.000, C 0.000 }
gfCNCPoint1[6445] = {X 296.2131, Y 100.7434, Z -1.3333, A 0.000, B 0.000, C 0.000 }
gfCNCPoint1[6446] = {X 295.5164, Y 101.4401, Z -1.3333, A 0.000, B 0.000, C 0.000 }
gfCNCPoint1[6447] = {X 294.6822, Y 101.9643, Z -1.3333, A 0.000, B 0.000, C 0.000 }
gfCNCPoint1[6448] = {X 293.7522, Y 102.2897, Z -1.3333, A 0.000, B 0.000, C 0.000 }
gfCNCPoint1[6449] = {X 292.7731, Y 102.4000, Z -1.3333, A 0.000, B 0.000, C 0.000 }
gfCNCPoint1[6450] = {X 276.2327, Y 102.4000, Z -1.3333, A 0.000, B 0.000, C 0.000 }
gfCNCPoint1[6451] = {X 275.2536, Y 102.2897, Z -1.3333, A 0.000, B 0.000, C 0.000 }
gfCNCPoint1[6452] = {X 274.3236, Y 101.9643, Z -1.3333, A 0.000, B 0.000, C 0.000 }
gfCNCPoint1[6453] = {X 273.4893, Y 101.4401, Z -1.3333, A 0.000, B 0.000, C 0.000 }
gfCNCPoint1[6454] = {X 272.7926, Y 100.7434, Z -1.3333, A 0.000, B 0.000, C 0.000 }
gfCNCPoint1[6455] = {X 272.2684, Y 99.9091, Z -1.3333, A 0.000, B 0.000, C 0.000 }
gfCNCPoint1[6456] = {X 271.9430, Y 98.9791, Z -1.3333, A 0.000, B 0.000, C 0.000 }
gfCNCPoint1[6457] = {X 271.8327, Y 98.0000, Z -1.3333, A 0.000, B 0.000, C 0.000 }
gfCNCPoint1[6458] = {X 271.8329, Y 97.0190, Z -1.3333, A 0.000, B 0.000, C 0.000 }
gfCNCPoint1[6459] = {X 271.9305, Y 96.1432, Z -1.3333, A 0.000, B 0.000, C 0.000 }
gfCNCPoint1[6460] = {X 272.2006, Y 95.3045, Z -1.3333, A 0.000, B 0.000, C 0.000 }
gfCNCPoint1[6461] = {X 272.6325, Y 94.5364, Z -1.3333, A 0.000, B 0.000, C 0.000 }
gfCNCPoint1[6462] = {X 273.2087, Y 93.8698, Z -1.3333, A 0.000, B 0.000, C 0.000 }
gfCNCPoint1[6463] = {X 273.9062, Y 93.3313, Z -1.3333, A 0.000, B 0.000, C 0.000 }
gfCNCPoint1[6464] = {X 274.6970, Y 92.9426, Z -1.3333, A 0.000, B 0.000, C 0.000 }
gfCNCPoint1[6465] = {X 275.5494, Y 92.7193, Z -1.3333, A 0.000, B 0.000, C 0.000 }
gfCNCPoint1[6466] = {X 275.5494, Y 85.6495, Z -1.3333, A 0.000, B 0.000, C 0.000 }
gfCNCPoint1[6467] = {X 262.6479, Y 80.5921, Z -1.3333, A 0.000, B 0.000, C 0.000 }
gfCNCPoint1[6468] = {X 262.3186, Y 80.7992, Z -1.3333, A 0.000, B 0.000, C 0.000 }
gfCNCPoint1[6469] = {X 237.8761, Y 96.6311, Z -1.3333, A 0.000, B 0.000, C 0.000 }
gfCNCPoint1[6470] = {X 237.8798, Y 97.0659, Z -1.3333, A 0.000, B 0.000, C 0.000 }
gfCNCPoint1[6471] = {X 237.8798, Y 98.0000, Z -1.3333, A 0.000, B 0.000, C 0.000 }
gfCNCPoint1[6472] = {X 237.7695, Y 98.9791, Z -1.3333, A 0.000, B 0.000, C 0.000 }
gfCNCPoint1[6473] = {X 237.4440, Y 99.9091, Z -1.3333, A 0.000, B 0.000, C 0.000 }
gfCNCPoint1[6474] = {X 236.9198, Y 100.7434, Z -1.3333, A 0.000, B 0.000, C 0.000 }
gfCNCPoint1[6475] = {X 236.2231, Y 101.4401, Z -1.3333, A 0.000, B 0.000, C 0.000 }
gfCNCPoint1[6476] = {X 235.3889, Y 101.9643, Z -1.3333, A 0.000, B 0.000, C 0.000 }
gfCNCPoint1[6477] = {X 234.4589, Y 102.2897, Z -1.3333, A 0.000, B 0.000, C 0.000 }
gfCNCPoint1[6478] = {X 233.4798, Y 102.4000, Z -1.3333, A 0.000, B 0.000, C 0.000 }
gfCNCPoint1[6479] = {X 214.1790, Y 102.4000, Z -1.3333, A 0.000, B 0.000, C 0.000 }
gfCNCPoint1[6480] = {X 213.7862, Y 102.3824, Z -1.3333, A 0.000, B 0.000, C 0.000 }
gfCNCPoint1[6481] = {X 213.3966, Y 102.3299, Z -1.3333, A 0.000, B 0.000, C 0.000 }
gfCNCPoint1[6482] = {X 213.0069, Y 102.3824, Z -1.3333, A 0.000, B 0.000, C 0.000 }
gfCNCPoint1[6483] = {X 212.6141, Y 102.4000, Z -1.3333, A 0.000, B 0.000, C 0.000 }
gfCNCPoint1[6484] = {X 194.9870, Y 102.4000, Z -1.3333, A 0.000, B 0.000, C 0.000 }
gfCNCPoint1[6485] = {X 194.0079, Y 102.2897, Z -1.3333, A 0.000, B 0.000, C 0.000 }
gfCNCPoint1[6486] = {X 193.0779, Y 101.9643, Z -1.3333, A 0.000, B 0.000, C 0.000 }
gfCNCPoint1[6487] = {X 192.2436, Y 101.4401, Z -1.3333, A 0.000, B 0.000, C 0.000 }
gfCNCPoint1[6488] = {X 191.5469, Y 100.7434, Z -1.3333, A 0.000, B 0.000, C 0.000 }
gfCNCPoint1[6489] = {X 191.0227, Y 99.9091, Z -1.3333, A 0.000, B 0.000, C 0.000 }
gfCNCPoint1[6490] = {X 190.6973, Y 98.9791, Z -1.3333, A 0.000, B 0.000, C 0.000 }
gfCNCPoint1[6491] = {X 190.5870, Y 98.0000, Z -1.3333, A 0.000, B 0.000, C 0.000 }
gfCNCPoint1[6492] = {X 190.5870, Y 97.0659, Z -1.3333, A 0.000, B 0.000, C 0.000 }
gfCNCPoint1[6493] = {X 190.6897, Y 96.1207, Z -1.3333, A 0.000, B 0.000, C 0.000 }
gfCNCPoint1[6494] = {X 190.9931, Y 95.2196, Z -1.3333, A 0.000, B 0.000, C 0.000 }
gfCNCPoint1[6495] = {X 191.4830, Y 94.4047, Z -1.3333, A 0.000, B 0.000, C 0.000 }
gfCNCPoint1[6496] = {X 188.5295, Y 91.1802, Z -1.3333, A 0.000, B 0.000, C 0.000 }
gfCNCPoint1[6497] = {X 150.1254, Y 91.1802, Z -1.3333, A 0.000, B 0.000, C 0.000 }
gfCNCPoint1[6498] = {X 147.2489, Y 94.3670, Z -1.3333, A 0.000, B 0.000, C 0.000 }
gfCNCPoint1[6499] = {X 147.7548, Y 95.1911, Z -1.3333, A 0.000, B 0.000, C 0.000 }
gfCNCPoint1[6500] = {X 148.0698, Y 96.1053, Z -1.3333, A 0.000, B 0.000, C 0.000 }
gfCNCPoint1[6501] = {X 148.1791, Y 97.0661, Z -1.3333, A 0.000, B 0.000, C 0.000 }
gfCNCPoint1[6502] = {X 148.1791, Y 98.0000, Z -1.3333, A 0.000, B 0.000, C 0.000 }
gfCNCPoint1[6503] = {X 148.0688, Y 98.9791, Z -1.3333, A 0.000, B 0.000, C 0.000 }
gfCNCPoint1[6504] = {X 147.7434, Y 99.9091, Z -1.3333, A 0.000, B 0.000, C 0.000 }
gfCNCPoint1[6505] = {X 147.2192, Y 100.7434, Z -1.3333, A 0.000, B 0.000, C 0.000 }
gfCNCPoint1[6506] = {X 146.5225, Y 101.4401, Z -1.3333, A 0.000, B 0.000, C 0.000 }
gfCNCPoint1[6507] = {X 145.6882, Y 101.9643, Z -1.3333, A 0.000, B 0.000, C 0.000 }
gfCNCPoint1[6508] = {X 144.7582, Y 102.2897, Z -1.3333, A 0.000, B 0.000, C 0.000 }
gfCNCPoint1[6509] = {X 143.7791, Y 102.4000, Z -1.3333, A 0.000, B 0.000, C 0.000 }
gfCNCPoint1[6510] = {X 125.0000, Y 102.4000, Z -1.3333, A 0.000, B 0.000, C 0.000 }
gfCNCPoint1[6511] = {X 124.0209, Y 102.2897, Z -1.3333, A 0.000, B 0.000, C 0.000 }
gfCNCPoint1[6512] = {X 123.0909, Y 101.9643, Z -1.3333, A 0.000, B 0.000, C 0.000 }
gfCNCPoint1[6513] = {X 122.2566, Y 101.4401, Z -1.3333, A 0.000, B 0.000, C 0.000 }
gfCNCPoint1[6514] = {X 121.5599, Y 100.7434, Z -1.3333, A 0.000, B 0.000, C 0.000 }
gfCNCPoint1[6515] = {X 121.0357, Y 99.9091, Z -1.3333, A 0.000, B 0.000, C 0.000 }
gfCNCPoint1[6516] = {X 120.7103, Y 98.9791, Z -1.3333, A 0.000, B 0.000, C 0.000 }
gfCNCPoint1[6517] = {X 120.6000, Y 98.0000, Z -1.3333, A 0.000, B 0.000, C 0.000 }
gfCNCPoint1[6518] = {X 120.6000, Y 97.0659, Z -1.3333, A 0.000, B 0.000, C 0.000 }
gfCNCPoint1[6519] = {X 120.7047, Y 96.1116, Z -1.3333, A 0.000, B 0.000, C 0.000 }
gfCNCPoint1[6520] = {X 121.0140, Y 95.2027, Z -1.3333, A 0.000, B 0.000, C 0.000 }
gfCNCPoint1[6521] = {X 121.5130, Y 94.3825, Z -1.3333, A 0.000, B 0.000, C 0.000 }
gfCNCPoint1[6522] = {X 122.1781, Y 93.6900, Z -1.3333, A 0.000, B 0.000, C 0.000 }
gfCNCPoint1[6523] = {X 122.9775, Y 93.1583, Z -1.3333, A 0.000, B 0.000, C 0.000 }
gfCNCPoint1[6524] = {X 123.8732, Y 92.8127, Z -1.3333, A 0.000, B 0.000, C 0.000 }
gfCNCPoint1[6525] = {X 124.8226, Y 92.6695, Z -1.3333, A 0.000, B 0.000, C 0.000 }
gfCNCPoint1[6526] = {X 124.8686, Y 92.6537, Z -1.3333, A 0.000, B 0.000, C 0.000 }
gfCNCPoint1[6527] = {X 124.9163, Y 92.6437, Z -1.3333, A 0.000, B 0.000, C 0.000 }
gfCNCPoint1[6528] = {X 125.4404, Y 92.5659, Z -1.3333, A 0.000, B 0.000, C 0.000 }
gfCNCPoint1[6529] = {X 126.2565, Y 92.4280, Z -1.3333, A 0.000, B 0.000, C 0.000 }
gfCNCPoint1[6530] = {X 127.0617, Y 92.2366, Z -1.3333, A 0.000, B 0.000, C 0.000 }
gfCNCPoint1[6531] = {X 128.2735, Y 91.0928, Z -1.3333, A 0.000, B 0.000, C 0.000 }
gfCNCPoint1[6532] = {X 129.4220, Y 89.8854, Z -1.3333, A 0.000, B 0.000, C 0.000 }
gfCNCPoint1[6533] = {X 133.5081, Y 85.3905, Z -1.3333, A 0.000, B 0.000, C 0.000 }
gfCNCPoint1[6534] = {X 155.5333, Y 61.2116, Z -1.3333, A 0.000, B 0.000, C 0.000 }
gfCNCPoint1[6535] = {X 155.1842, Y 60.4953, Z -1.3333, A 0.000, B 0.000, C 0.000 }
gfCNCPoint1[6536] = {X 154.9701, Y 59.7277, Z -1.3333, A 0.000, B 0.000, C 0.000 }
gfCNCPoint1[6537] = {X 154.8980, Y 58.9340, Z -1.3333, A 0.000, B 0.000, C 0.000 }
gfCNCPoint1[6538] = {X 154.8980, Y 58.0000, Z -1.3333, A 0.000, B 0.000, C 0.000 }
gfCNCPoint1[6539] = {X 155.0083, Y 57.0209, Z -1.3333, A 0.000, B 0.000, C 0.000 }
gfCNCPoint1[6540] = {X 155.3337, Y 56.0909, Z -1.3333, A 0.000, B 0.000, C 0.000 }
gfCNCPoint1[6541] = {X 155.8579, Y 55.2566, Z -1.3333, A 0.000, B 0.000, C 0.000 }
gfCNCPoint1[6542] = {X 156.5546, Y 54.5599, Z -1.3333, A 0.000, B 0.000, C 0.000 }
gfCNCPoint1[6543] = {X 157.3889, Y 54.0357, Z -1.3333, A 0.000, B 0.000, C 0.000 }
gfCNCPoint1[6544] = {X 158.3189, Y 53.7103, Z -1.3333, A 0.000, B 0.000, C 0.000 }
gfCNCPoint1[6545] = {X 159.2980, Y 53.6000, Z -1.3333, A 0.000, B 0.000, C 0.000 }
gfCNCPoint1[6546] = {X 178.5335, Y 53.6000, Z -1.3333, A 0.000, B 0.000, C 0.000 }
gfCNCPoint1[6547] = {X 179.5126, Y 53.7103, Z -1.3333, A 0.000, B 0.000, C 0.000 }
gfCNCPoint1[6548] = {X 180.4426, Y 54.0357, Z -1.3333, A 0.000, B 0.000, C 0.000 }
gfCNCPoint1[6549] = {X 181.2769, Y 54.5599, Z -1.3333, A 0.000, B 0.000, C 0.000 }
gfCNCPoint1[6550] = {X 181.9736, Y 55.2566, Z -1.3333, A 0.000, B 0.000, C 0.000 }
gfCNCPoint1[6551] = {X 182.4978, Y 56.0909, Z -1.3333, A 0.000, B 0.000, C 0.000 }
gfCNCPoint1[6552] = {X 182.8232, Y 57.0209, Z -1.3333, A 0.000, B 0.000, C 0.000 }
gfCNCPoint1[6553] = {X 182.9335, Y 58.0000, Z -1.3333, A 0.000, B 0.000, C 0.000 }
gfCNCPoint1[6554] = {X 182.9334, Y 58.9704, Z -1.3333, A 0.000, B 0.000, C 0.000 }
gfCNCPoint1[6555] = {X 182.8587, Y 59.7421, Z -1.3333, A 0.000, B 0.000, C 0.000 }
gfCNCPoint1[6556] = {X 182.6497, Y 60.4888, Z -1.3333, A 0.000, B 0.000, C 0.000 }
gfCNCPoint1[6557] = {X 182.3129, Y 61.1872, Z -1.3333, A 0.000, B 0.000, C 0.000 }
gfCNCPoint1[6558] = {X 209.5361, Y 90.8997, Z -1.3333, A 0.000, B 0.000, C 0.000 }
gfCNCPoint1[6559] = {X 210.1905, Y 91.5636, Z -1.3333, A 0.000, B 0.000, C 0.000 }
gfCNCPoint1[6560] = {X 210.8914, Y 92.1781, Z -1.3333, A 0.000, B 0.000, C 0.000 }
gfCNCPoint1[6561] = {X 211.1540, Y 92.3434, Z -1.3333, A 0.000, B 0.000, C 0.000 }
gfCNCPoint1[6562] = {X 211.4487, Y 92.4406, Z -1.3333, A 0.000, B 0.000, C 0.000 }
gfCNCPoint1[6563] = {X 212.4320, Y 92.6229, Z -1.3333, A 0.000, B 0.000, C 0.000 }
gfCNCPoint1[6564] = {X 213.4256, Y 92.7359, Z -1.3333, A 0.000, B 0.000, C 0.000 }
gfCNCPoint1[6565] = {X 214.4671, Y 92.6568, Z -1.3333, A 0.000, B 0.000, C 0.000 }
gfCNCPoint1[6566] = {X 215.5098, Y 92.5968, Z -1.3333, A 0.000, B 0.000, C 0.000 }
gfCNCPoint1[6567] = {X 216.1639, Y 92.5246, Z -1.3333, A 0.000, B 0.000, C 0.000 }
gfCNCPoint1[6568] = {X 216.7936, Y 92.3339, Z -1.3333, A 0.000, B 0.000, C 0.000 }
gfCNCPoint1[6569] = {X 217.3779, Y 92.0310, Z -1.3333, A 0.000, B 0.000, C 0.000 }
gfCNCPoint1[6570] = {X 222.9188, Y 88.4552, Z -1.3333, A 0.000, B 0.000, C 0.000 }
gfCNCPoint1[6571] = {X 245.6542, Y 73.9166, Z -1.3333, A 0.000, B 0.000, C 0.000 }
gfCNCPoint1[6572] = {X 221.6008, Y 64.4767, Z -1.3333, A 0.000, B 0.000, C 0.000 }
gfCNCPoint1[6573] = {X 219.8423, Y 63.8881, Z -1.3333, A 0.000, B 0.000, C 0.000 }
gfCNCPoint1[6574] = {X 218.0280, Y 63.5047, Z -1.3333, A 0.000, B 0.000, C 0.000 }
gfCNCPoint1[6575] = {X 216.1818, Y 63.3315, Z -1.3333, A 0.000, B 0.000, C 0.000 }
gfCNCPoint1[6576] = {X 215.2276, Y 63.1935, Z -1.3333, A 0.000, B 0.000, C 0.000 }
gfCNCPoint1[6577] = {X 214.3264, Y 62.8510, Z -1.3333, A 0.000, B 0.000, C 0.000 }
gfCNCPoint1[6578] = {X 213.5214, Y 62.3204, Z -1.3333, A 0.000, B 0.000, C 0.000 }
gfCNCPoint1[6579] = {X 212.8513, Y 61.6272, Z -1.3333, A 0.000, B 0.000, C 0.000 }
gfCNCPoint1[6580] = {X 212.3482, Y 60.8047, Z -1.3333, A 0.000, B 0.000, C 0.000 }
gfCNCPoint1[6581] = {X 212.0364, Y 59.8924, Z -1.3333, A 0.000, B 0.000, C 0.000 }
gfCNCPoint1[6582] = {X 211.9308, Y 58.9340, Z -1.3333, A 0.000, B 0.000, C 0.000 }
gfCNCPoint1[6583] = {X 211.9308, Y 58.0000, Z -1.3333, A 0.000, B 0.000, C 0.000 }
gfCNCPoint1[6584] = {X 212.0411, Y 57.0209, Z -1.3333, A 0.000, B 0.000, C 0.000 }
gfCNCPoint1[6585] = {X 212.3665, Y 56.0909, Z -1.3333, A 0.000, B 0.000, C 0.000 }
gfCNCPoint1[6586] = {X 212.8907, Y 55.2566, Z -1.3333, A 0.000, B 0.000, C 0.000 }
gfCNCPoint1[6587] = {X 213.5875, Y 54.5599, Z -1.3333, A 0.000, B 0.000, C 0.000 }
gfCNCPoint1[6588] = {X 214.4217, Y 54.0357, Z -1.3333, A 0.000, B 0.000, C 0.000 }
gfCNCPoint1[6589] = {X 215.3517, Y 53.7103, Z -1.3333, A 0.000, B 0.000, C 0.000 }
gfCNCPoint1[6590] = {X 216.3308, Y 53.6000, Z -1.3333, A 0.000, B 0.000, C 0.000 }
gfCNCPoint1[6591] = {X 237.2617, Y 53.6000, Z -1.3333, A 0.000, B 0.000, C 0.000 }
gfCNCPoint1[6592] = {X 238.2408, Y 53.7103, Z -1.3333, A 0.000, B 0.000, C 0.000 }
gfCNCPoint1[6593] = {X 239.1708, Y 54.0357, Z -1.3333, A 0.000, B 0.000, C 0.000 }
gfCNCPoint1[6594] = {X 240.0050, Y 54.5599, Z -1.3333, A 0.000, B 0.000, C 0.000 }
gfCNCPoint1[6595] = {X 240.7017, Y 55.2566, Z -1.3333, A 0.000, B 0.000, C 0.000 }
gfCNCPoint1[6596] = {X 241.2260, Y 56.0909, Z -1.3333, A 0.000, B 0.000, C 0.000 }
gfCNCPoint1[6597] = {X 241.5514, Y 57.0209, Z -1.3333, A 0.000, B 0.000, C 0.000 }
gfCNCPoint1[6598] = {X 241.6617, Y 58.0000, Z -1.3333, A 0.000, B 0.000, C 0.000 }
gfCNCPoint1[6599] = {X 241.6617, Y 58.1784, Z -1.3333, A 0.000, B 0.000, C 0.000 }
gfCNCPoint1[6600] = {X 248.1429, Y 60.7053, Z -1.3333, A 0.000, B 0.000, C 0.000 }
gfCNCPoint1[6601] = {X 275.5541, Y 71.5853, Z -1.3333, A 0.000, B 0.000, C 0.000 }
gfCNCPoint1[6602] = {X 275.5533, Y 63.2813, Z -1.3333, A 0.000, B 0.000, C 0.000 }
gfCNCPoint1[6603] = {X 274.6939, Y 63.0562, Z -1.3333, A 0.000, B 0.000, C 0.000 }
gfCNCPoint1[6604] = {X 273.8972, Y 62.6631, Z -1.3333, A 0.000, B 0.000, C 0.000 }
gfCNCPoint1[6605] = {X 273.1957, Y 62.1179, Z -1.3333, A 0.000, B 0.000, C 0.000 }
gfCNCPoint1[6606] = {X 272.6181, Y 61.4430, Z -1.3333, A 0.000, B 0.000, C 0.000 }
gfCNCPoint1[6607] = {X 272.1878, Y 60.6657, Z -1.3333, A 0.000, B 0.000, C 0.000 }
gfCNCPoint1[6608] = {X 271.9224, Y 59.8179, Z -1.3333, A 0.000, B 0.000, C 0.000 }
gfCNCPoint1[6609] = {X 271.8327, Y 58.9340, Z -1.3333, A 0.000, B 0.000, C 0.000 }
gfCNCPoint1[6610] = {X 271.8327, Y 58.0000, Z -1.3333, A 0.000, B 0.000, C 0.000 }
gfCNCPoint1[6611] = {X 271.9430, Y 57.0209, Z -1.3333, A 0.000, B 0.000, C 0.000 }
gfCNCPoint1[6612] = {X 272.2684, Y 56.0909, Z -1.3333, A 0.000, B 0.000, C 0.000 }
gfCNCPoint1[6613] = {X 272.7926, Y 55.2566, Z -1.3333, A 0.000, B 0.000, C 0.000 }
gfCNCPoint1[6614] = {X 273.4893, Y 54.5599, Z -1.3333, A 0.000, B 0.000, C 0.000 }
gfCNCPoint1[6615] = {X 274.3236, Y 54.0357, Z -1.3333, A 0.000, B 0.000, C 0.000 }
gfCNCPoint1[6616] = {X 275.2536, Y 53.7103, Z -1.3333, A 0.000, B 0.000, C 0.000 }
gfCNCPoint1[6617] = {X 276.2327, Y 53.6000, Z -1.3333, A 0.000, B 0.000, C 0.000 }
gfCNCPoint1[6618] = {X 292.7731, Y 53.6000, Z -1.3333, A 0.000, B 0.000, C 0.000 }
gfCNCPoint1[6619] = {X 293.7522, Y 53.7103, Z -1.3333, A 0.000, B 0.000, C 0.000 }
gfCNCPoint1[6620] = {X 294.6822, Y 54.0357, Z -1.3333, A 0.000, B 0.000, C 0.000 }
gfCNCPoint1[6621] = {X 295.5164, Y 54.5599, Z -1.3333, A 0.000, B 0.000, C 0.000 }
gfCNCPoint1[6622] = {X 296.2131, Y 55.2566, Z -1.3333, A 0.000, B 0.000, C 0.000 }
gfCNCPoint1[6623] = {X 296.7373, Y 56.0909, Z -1.3333, A 0.000, B 0.000, C 0.000 }
gfCNCPoint1[6624] = {X 297.0628, Y 57.0209, Z -1.3333, A 0.000, B 0.000, C 0.000 }
gfCNCPoint1[6625] = {X 297.1731, Y 58.0000, Z -1.3333, A 0.000, B 0.000, C 0.000 }
gfCNCPoint1[6626] = {X 297.1731, Y 58.9355, Z -1.3333, A 0.000, B 0.000, C 0.000 }
gfCNCPoint1[6627] = {X 297.0807, Y 59.8184, Z -1.3333, A 0.000, B 0.000, C 0.000 }
gfCNCPoint1[6628] = {X 296.8137, Y 60.6649, Z -1.3333, A 0.000, B 0.000, C 0.000 }
gfCNCPoint1[6629] = {X 296.3828, Y 61.4410, Z -1.3333, A 0.000, B 0.000, C 0.000 }
gfCNCPoint1[6630] = {X 295.8055, Y 62.1153, Z -1.3333, A 0.000, B 0.000, C 0.000 }
gfCNCPoint1[6631] = {X 295.1049, Y 62.6605, Z -1.3333, A 0.000, B 0.000, C 0.000 }
gfCNCPoint1[6632] = {X 294.3096, Y 63.0546, Z -1.3333, A 0.000, B 0.000, C 0.000 }
gfCNCPoint1[6633] = {X 293.4514, Y 63.2817, Z -1.3333, A 0.000, B 0.000, C 0.000 }
gfCNCPoint1[6634] = {X 293.4514, Y 92.7120, Z -1.3333, A 0.000, B 0.000, C 0.000 }
gfCNCPoint1[6635] = {X 294.3094, Y 92.9416, Z -1.3333, A 0.000, B 0.000, C 0.000 }
gfCNCPoint1[6636] = {X 295.1044, Y 93.3376, Z -1.3333, A 0.000, B 0.000, C 0.000 }
gfCNCPoint1[6637] = {X 295.8044, Y 93.8842, Z -1.3333, A 0.000, B 0.000, C 0.000 }
gfCNCPoint1[6638] = {X 296.3815, Y 94.5593, Z -1.3333, A 0.000, B 0.000, C 0.000 }
gfCNCPoint1[6639] = {X 296.8124, Y 95.3360, Z -1.3333, A 0.000, B 0.000, C 0.000 }
gfCNCPoint1[6640] = {X 297.0798, Y 96.1829, Z -1.3333, A 0.000, B 0.000, C 0.000 }
gfCNCPoint1[6641] = {X 297.1731, Y 97.0661, Z -1.3333, A 0.000, B 0.000, C 0.000 }
gfCNCPoint1[6642] = {X 297.1731, Y 97.6949, Z -1.3333, A 0.000, B 0.000, C 0.000 }
gfCNCPoint1[6643] = {X 297.6531, Y 97.6949, Z -1.3333, A 0.000, B 0.000, C 0.000 }
gfCNCPoint1[6644] = {X 314.2131, Y 97.6949, Z -1.3333, A 0.000, B 0.000, C 0.000 }
gfCNCPoint1[6645] = {X 313.0151, Y 96.8440, Z -1.3333, A 0.000, B 0.000, C 0.000 }
gfCNCPoint1[6646] = {X 311.8814, Y 95.9090, Z -1.3333, A 0.000, B 0.000, C 0.000 }
gfCNCPoint1[6647] = {X 310.9068, Y 94.9477, Z -1.3333, A 0.000, B 0.000, C 0.000 }
gfCNCPoint1[6648] = {X 310.0433, Y 93.8854, Z -1.3333, A 0.000, B 0.000, C 0.000 }
gfCNCPoint1[6649] = {X 309.2093, Y 92.5708, Z -1.3333, A 0.000, B 0.000, C 0.000 }
gfCNCPoint1[6650] = {X 308.5454, Y 91.1626, Z -1.3333, A 0.000, B 0.000, C 0.000 }
gfCNCPoint1[6651] = {X 308.0619, Y 89.6827, Z -1.3333, A 0.000, B 0.000, C 0.000 }
gfCNCPoint1[6652] = {X 307.7084, Y 88.0127, Z -1.3333, A 0.000, B 0.000, C 0.000 }
gfCNCPoint1[6653] = {X 307.4995, Y 86.3185, Z -1.3333, A 0.000, B 0.000, C 0.000 }
gfCNCPoint1[6654] = {X 307.4367, Y 84.6126, Z -1.3333, A 0.000, B 0.000, C 0.000 }
gfCNCPoint1[6655] = {X 307.4380, Y 83.2305, Z -1.3333, A 0.000, B 0.000, C 0.000 }
gfCNCPoint1[6656] = {X 307.4380, Y 63.6746, Z -1.3333, A 0.000, B 0.000, C 0.000 }
gfCNCPoint1[6657] = {X 306.4292, Y 63.3065, Z -1.3333, A 0.000, B 0.000, C 0.000 }
gfCNCPoint1[6658] = {X 305.5254, Y 62.7268, Z -1.3333, A 0.000, B 0.000, C 0.000 }
gfCNCPoint1[6659] = {X 304.7703, Y 61.9634, Z -1.3333, A 0.000, B 0.000, C 0.000 }
gfCNCPoint1[6660] = {X 304.2004, Y 61.0533, Z -1.3333, A 0.000, B 0.000, C 0.000 }
gfCNCPoint1[6661] = {X 303.8433, Y 60.0406, Z -1.3333, A 0.000, B 0.000, C 0.000 }
gfCNCPoint1[6662] = {X 303.7164, Y 58.9744, Z -1.3333, A 0.000, B 0.000, C 0.000 }
gfCNCPoint1[6663] = {X 303.7162, Y 58.0000, Z -1.3333, A 0.000, B 0.000, C 0.000 }
gfCNCPoint1[6664] = {X 303.8100, Y 57.0480, Z -1.3333, A 0.000, B 0.000, C 0.000 }
gfCNCPoint1[6665] = {X 304.0877, Y 56.1325, Z -1.3333, A 0.000, B 0.000, C 0.000 }
gfCNCPoint1[6666] = {X 304.5387, Y 55.2888, Z -1.3333, A 0.000, B 0.000, C 0.000 }
gfCNCPoint1[6667] = {X 305.1455, Y 54.5493, Z -1.3333, A 0.000, B 0.000, C 0.000 }
gfCNCPoint1[6668] = {X 305.8850, Y 53.9424, Z -1.3333, A 0.000, B 0.000, C 0.000 }
gfCNCPoint1[6669] = {X 306.7287, Y 53.4915, Z -1.3333, A 0.000, B 0.000, C 0.000 }
gfCNCPoint1[6670] = {X 307.6442, Y 53.2138, Z -1.3333, A 0.000, B 0.000, C 0.000 }
gfCNCPoint1[6671] = {X 308.5962, Y 53.1200, Z -1.3333, A 0.000, B 0.000, C 0.000 }
gfCNCPoint1[6672] = {X 324.3107, Y 53.1200, Z -1.3333, A 0.000, B 0.000, C 0.000 }
gfCNCPoint1[6673] = {X 325.2627, Y 53.2138, Z -1.3333, A 0.000, B 0.000, C 0.000 }
gfCNCPoint1[6674] = {X 326.1782, Y 53.4915, Z -1.3333, A 0.000, B 0.000, C 0.000 }
gfCNCPoint1[6675] = {X 327.0219, Y 53.9424, Z -1.3333, A 0.000, B 0.000, C 0.000 }
gfCNCPoint1[6676] = {X 327.7614, Y 54.5493, Z -1.3333, A 0.000, B 0.000, C 0.000 }
gfCNCPoint1[6677] = {X 328.3683, Y 55.2888, Z -1.3333, A 0.000, B 0.000, C 0.000 }
gfCNCPoint1[6678] = {X 328.8192, Y 56.1325, Z -1.3333, A 0.000, B 0.000, C 0.000 }
gfCNCPoint1[6679] = {X 329.0969, Y 57.0480, Z -1.3333, A 0.000, B 0.000, C 0.000 }
gfCNCPoint1[6680] = {X 329.1907, Y 58.0000, Z -1.3333, A 0.000, B 0.000, C 0.000 }
gfCNCPoint1[6681] = {X 329.1907, Y 58.9341, Z -1.3333, A 0.000, B 0.000, C 0.000 }
gfCNCPoint1[6682] = {X 329.0667, Y 60.0066, Z -1.3333, A 0.000, B 0.000, C 0.000 }
gfCNCPoint1[6683] = {X 328.7117, Y 61.0262, Z -1.3333, A 0.000, B 0.000, C 0.000 }
gfCNCPoint1[6684] = {X 328.1430, Y 61.9438, Z -1.3333, A 0.000, B 0.000, C 0.000 }
gfCNCPoint1[6685] = {X 327.3877, Y 62.7153, Z -1.3333, A 0.000, B 0.000, C 0.000 }
gfCNCPoint1[6686] = {X 326.4824, Y 63.3035, Z -1.3333, A 0.000, B 0.000, C 0.000 }
gfCNCPoint1[6687] = {X 325.4706, Y 63.6801, Z -1.3333, A 0.000, B 0.000, C 0.000 }
gfCNCPoint1[6688] = {X 325.4719, Y 83.2268, Z -1.3333, A 0.000, B 0.000, C 0.000 }
gfCNCPoint1[6689] = {X 325.4854, Y 84.6073, Z -1.3333, A 0.000, B 0.000, C 0.000 }
gfCNCPoint1[6690] = {X 325.5512, Y 85.7203, Z -1.3333, A 0.000, B 0.000, C 0.000 }
gfCNCPoint1[6691] = {X 325.7422, Y 86.8187, Z -1.3333, A 0.000, B 0.000, C 0.000 }
gfCNCPoint1[6692] = {X 325.8861, Y 86.9531, Z -1.3333, A 0.000, B 0.000, C 0.000 }
gfCNCPoint1[6693] = {X 326.0542, Y 87.0555, Z -1.3333, A 0.000, B 0.000, C 0.000 }
gfCNCPoint1[6694] = {X 326.4824, Y 87.2970, Z -1.3333, A 0.000, B 0.000, C 0.000 }
gfCNCPoint1[6695] = {X 327.8560, Y 87.8663, Z -1.3333, A 0.000, B 0.000, C 0.000 }
gfCNCPoint1[6696] = {X 329.2836, Y 88.2819, Z -1.3333, A 0.000, B 0.000, C 0.000 }
gfCNCPoint1[6697] = {X 332.3214, Y 88.8903, Z -1.3333, A 0.000, B 0.000, C 0.000 }
gfCNCPoint1[6698] = {X 335.3951, Y 89.2777, Z -1.3333, A 0.000, B 0.000, C 0.000 }
gfCNCPoint1[6699] = {X 340.5456, Y 89.6591, Z -1.3333, A 0.000, B 0.000, C 0.000 }
gfCNCPoint1[6700] = {X 345.7083, Y 89.8032, Z -1.3333, A 0.000, B 0.000, C 0.000 }
gfCNCPoint1[6701] = {X 350.5332, Y 89.8095, Z -1.3333, A 0.000, B 0.000, C 0.000 }
gfCNCPoint1[6702] = {X 355.3552, Y 89.6417, Z -1.3333, A 0.000, B 0.000, C 0.000 }
gfCNCPoint1[6703] = {X 360.1680, Y 89.3003, Z -1.3333, A 0.000, B 0.000, C 0.000 }
gfCNCPoint1[6704] = {X 362.6809, Y 89.0151, Z -1.3333, A 0.000, B 0.000, C 0.000 }
gfCNCPoint1[6705] = {X 365.1707, Y 88.5712, Z -1.3333, A 0.000, B 0.000, C 0.000 }
gfCNCPoint1[6706] = {X 367.6273, Y 87.9701, Z -1.3333, A 0.000, B 0.000, C 0.000 }
gfCNCPoint1[6707] = {X 368.9202, Y 87.4951, Z -1.3333, A 0.000, B 0.000, C 0.000 }
gfCNCPoint1[6708] = {X 370.1152, Y 86.8102, Z -1.3333, A 0.000, B 0.000, C 0.000 }
gfCNCPoint1[6709] = {X 370.2998, Y 85.3240, Z -1.3333, A 0.000, B 0.000, C 0.000 }
gfCNCPoint1[6710] = {X 370.3614, Y 83.8277, Z -1.3333, A 0.000, B 0.000, C 0.000 }
gfCNCPoint1[6711] = {X 370.3597, Y 63.6743, Z -1.3333, A 0.000, B 0.000, C 0.000 }
gfCNCPoint1[6712] = {X 369.3513, Y 63.3060, Z -1.3333, A 0.000, B 0.000, C 0.000 }
gfCNCPoint1[6713] = {X 368.4478, Y 62.7262, Z -1.3333, A 0.000, B 0.000, C 0.000 }
gfCNCPoint1[6714] = {X 367.6929, Y 61.9628, Z -1.3333, A 0.000, B 0.000, C 0.000 }
gfCNCPoint1[6715] = {X 367.1233, Y 61.0529, Z -1.3333, A 0.000, B 0.000, C 0.000 }
gfCNCPoint1[6716] = {X 366.7663, Y 60.0404, Z -1.3333, A 0.000, B 0.000, C 0.000 }
gfCNCPoint1[6717] = {X 366.6394, Y 58.9744, Z -1.3333, A 0.000, B 0.000, C 0.000 }
gfCNCPoint1[6718] = {X 366.6393, Y 58.0000, Z -1.3333, A 0.000, B 0.000, C 0.000 }
gfCNCPoint1[6719] = {X 366.7331, Y 57.0480, Z -1.3333, A 0.000, B 0.000, C 0.000 }
gfCNCPoint1[6720] = {X 367.0108, Y 56.1325, Z -1.3333, A 0.000, B 0.000, C 0.000 }
gfCNCPoint1[6721] = {X 367.4617, Y 55.2888, Z -1.3333, A 0.000, B 0.000, C 0.000 }
gfCNCPoint1[6722] = {X 368.0686, Y 54.5493, Z -1.3333, A 0.000, B 0.000, C 0.000 }
gfCNCPoint1[6723] = {X 368.8081, Y 53.9424, Z -1.3333, A 0.000, B 0.000, C 0.000 }
gfCNCPoint1[6724] = {X 369.6518, Y 53.4915, Z -1.3333, A 0.000, B 0.000, C 0.000 }
gfCNCPoint1[6725] = {X 370.5672, Y 53.2138, Z -1.3333, A 0.000, B 0.000, C 0.000 }
gfCNCPoint1[6726] = {X 371.5193, Y 53.1200, Z -1.3333, A 0.000, B 0.000, C 0.000 }
gfCNCPoint1[6727] = {X 388.0597, Y 53.1200, Z -1.3333, A 0.000, B 0.000, C 0.000 }
gfCNCPoint1[6728] = {X 389.0355, Y 53.2186, Z -1.3333, A 0.000, B 0.000, C 0.000 }
gfCNCPoint1[6729] = {X 389.9719, Y 53.5102, Z -1.3333, A 0.000, B 0.000, C 0.000 }
gfCNCPoint1[6730] = {X 390.8310, Y 53.9833, Z -1.3333, A 0.000, B 0.000, C 0.000 }
gfCNCPoint1[6731] = {X 391.5783, Y 54.6186, Z -1.3333, A 0.000, B 0.000, C 0.000 }
gfCNCPoint1[6732] = {X 392.1572, Y 55.3496, Z -1.3333, A 0.000, B 0.000, C 0.000 }
gfCNCPoint1[6733] = {X 392.5865, Y 56.1774, Z -1.3333, A 0.000, B 0.000, C 0.000 }
gfCNCPoint1[6734] = {X 392.8506, Y 57.0718, Z -1.3333, A 0.000, B 0.000, C 0.000 }
gfCNCPoint1[6735] = {X 392.9397, Y 58.0000, Z -1.3333, A 0.000, B 0.000, C 0.000 }
gfCNCPoint1[6736] = {X 392.9395, Y 58.9744, Z -1.3333, A 0.000, B 0.000, C 0.000 }
gfCNCPoint1[6737] = {X 392.8769, Y 59.7141, Z -1.3333, A 0.000, B 0.000, C 0.000 }
gfCNCPoint1[6738] = {X 392.7029, Y 60.4358, Z -1.3333, A 0.000, B 0.000, C 0.000 }
gfCNCPoint1[6739] = {X 392.4214, Y 61.1227, Z -1.3333, A 0.000, B 0.000, C 0.000 }
gfCNCPoint1[6740] = {X 392.0443, Y 61.7518, Z -1.3333, A 0.000, B 0.000, C 0.000 }
gfCNCPoint1[6741] = {X 391.5775, Y 62.3176, Z -1.3333, A 0.000, B 0.000, C 0.000 }
gfCNCPoint1[6742] = {X 390.8815, Y 62.9184, Z -1.3333, A 0.000, B 0.000, C 0.000 }
gfCNCPoint1[6743] = {X 390.0856, Y 63.3786, Z -1.3333, A 0.000, B 0.000, C 0.000 }
gfCNCPoint1[6744] = {X 389.2176, Y 63.6821, Z -1.3333, A 0.000, B 0.000, C 0.000 }
gfCNCPoint1[6745] = {X 389.2167, Y 73.4803, Z -1.3333, A 0.000, B 0.000, C 0.000 }
gfCNCPoint1[6746] = {X 398.8167, Y 73.4812, Z -1.3333, A 0.000, B 0.000, C 0.000 }
gfCNCPoint1[6747] = {X 398.8160, Y 80.5599, Z -1.3333, A 0.000, B 0.000, C 0.000 }
gfCNCPoint1[6748] = {X 405.8059, Y 76.0831, Z -1.3333, A 0.000, B 0.000, C 0.000 }
gfCNCPoint1[6749] = {X 400.0357, Y 73.8191, Z -1.3333, A 0.000, B 0.000, C 0.000 }
gfCNCPoint1[6750] = {X 399.4350, Y 73.6183, Z -1.3333, A 0.000, B 0.000, C 0.000 }
gfCNCPoint1[6751] = {X 398.8167, Y 73.4812, Z -1.3333, A 0.000, B 0.000, C 0.000 }
gfCNCPoint1[6752] = {X 396.4167, Y 73.4810, Z -1.3333, A 0.000, B 0.000, C 0.000 }
gfCNCPoint1[6753] = {X 396.4156, Y 84.5902, Z -1.3333, A 0.000, B 0.000, C 0.000 }
gfCNCPoint1[6754] = {X 396.4154, Y 84.9474, Z -1.3333, A 0.000, B 0.000, C 0.000 }
gfCNCPoint1[6755] = {X 411.0615, Y 75.5672, Z -1.3333, A 0.000, B 0.000, C 0.000 }
gfCNCPoint1[6756] = {X 400.9145, Y 71.5857, Z -1.3333, A 0.000, B 0.000, C 0.000 }
gfCNCPoint1[6757] = {X 399.6214, Y 71.1929, Z -1.3333, A 0.000, B 0.000, C 0.000 }
gfCNCPoint1[6758] = {X 398.2823, Y 71.0109, Z -1.3333, A 0.000, B 0.000, C 0.000 }
gfCNCPoint1[6759] = {X 397.3460, Y 70.9531, Z -1.3333, A 0.000, B 0.000, C 0.000 }
gfCNCPoint1[6760] = {X 396.4169, Y 70.8229, Z -1.3333, A 0.000, B 0.000, C 0.000 }
gfCNCPoint1[6761] = {X 396.4167, Y 73.4810, Z -1.3333, A 0.000, B 0.000, C 0.000 }
gfCNCPoint1[6762] = {X 394.0167, Y 73.4808, Z -1.3333, A 0.000, B 0.000, C 0.000 }
gfCNCPoint1[6763] = {X 394.0156, Y 84.5977, Z -1.3333, A 0.000, B 0.000, C 0.000 }
gfCNCPoint1[6764] = {X 394.0161, Y 84.7640, Z -1.3333, A 0.000, B 0.000, C 0.000 }
gfCNCPoint1[6765] = {X 394.0155, Y 84.9302, Z -1.3333, A 0.000, B 0.000, C 0.000 }
gfCNCPoint1[6766] = {X 393.9650, Y 86.3347, Z -1.3333, A 0.000, B 0.000, C 0.000 }
gfCNCPoint1[6767] = {X 393.8336, Y 87.7340, Z -1.3333, A 0.000, B 0.000, C 0.000 }
gfCNCPoint1[6768] = {X 395.0700, Y 87.4786, Z -1.3333, A 0.000, B 0.000, C 0.000 }
gfCNCPoint1[6769] = {X 396.3291, Y 87.3862, Z -1.3333, A 0.000, B 0.000, C 0.000 }
gfCNCPoint1[6770] = {X 396.7234, Y 87.3732, Z -1.3333, A 0.000, B 0.000, C 0.000 }
gfCNCPoint1[6771] = {X 397.1171, Y 87.3480, Z -1.3333, A 0.000, B 0.000, C 0.000 }
gfCNCPoint1[6772] = {X 416.3171, Y 75.0512, Z -1.3333, A 0.000, B 0.000, C 0.000 }
gfCNCPoint1[6773] = {X 401.7933, Y 69.3524, Z -1.3333, A 0.000, B 0.000, C 0.000 }
gfCNCPoint1[6774] = {X 400.6815, Y 68.9829, Z -1.3333, A 0.000, B 0.000, C 0.000 }
gfCNCPoint1[6775] = {X 399.5364, Y 68.7352, Z -1.3333, A 0.000, B 0.000, C 0.000 }
gfCNCPoint1[6776] = {X 398.3713, Y 68.6123, Z -1.3333, A 0.000, B 0.000, C 0.000 }
gfCNCPoint1[6777] = {X 397.6038, Y 68.5669, Z -1.3333, A 0.000, B 0.000, C 0.000 }
gfCNCPoint1[6778] = {X 396.8423, Y 68.4608, Z -1.3333, A 0.000, B 0.000, C 0.000 }
gfCNCPoint1[6779] = {X 395.3918, Y 68.0817, Z -1.3333, A 0.000, B 0.000, C 0.000 }
gfCNCPoint1[6780] = {X 394.0173, Y 67.4831, Z -1.3333, A 0.000, B 0.000, C 0.000 }
gfCNCPoint1[6781] = {X 394.0167, Y 73.4808, Z -1.3333, A 0.000, B 0.000, C 0.000 }
gfCNCPoint1[6782] = {X 391.6167, Y 73.4805, Z -1.3333, A 0.000, B 0.000, C 0.000 }
gfCNCPoint1[6783] = {X 391.6156, Y 84.6056, Z -1.3333, A 0.000, B 0.000, C 0.000 }
gfCNCPoint1[6784] = {X 391.5794, Y 86.0259, Z -1.3333, A 0.000, B 0.000, C 0.000 }
gfCNCPoint1[6785] = {X 391.4516, Y 87.4409, Z -1.3333, A 0.000, B 0.000, C 0.000 }
gfCNCPoint1[6786] = {X 391.2273, Y 88.8722, Z -1.3333, A 0.000, B 0.000, C 0.000 }
gfCNCPoint1[6787] = {X 390.9093, Y 90.2857, Z -1.3333, A 0.000, B 0.000, C 0.000 }
gfCNCPoint1[6788] = {X 390.3333, Y 92.0497, Z -1.3333, A 0.000, B 0.000, C 0.000 }
gfCNCPoint1[6789] = {X 389.5419, Y 93.7281, Z -1.3333, A 0.000, B 0.000, C 0.000 }
gfCNCPoint1[6790] = {X 388.5476, Y 95.2949, Z -1.3333, A 0.000, B 0.000, C 0.000 }
gfCNCPoint1[6791] = {X 389.3447, Y 95.2949, Z -1.3333, A 0.000, B 0.000, C 0.000 }
gfCNCPoint1[6792] = {X 389.7639, Y 94.0858, Z -1.3333, A 0.000, B 0.000, C 0.000 }
gfCNCPoint1[6793] = {X 390.3884, Y 92.9687, Z -1.3333, A 0.000, B 0.000, C 0.000 }
gfCNCPoint1[6794] = {X 391.1988, Y 91.9783, Z -1.3333, A 0.000, B 0.000, C 0.000 }
gfCNCPoint1[6795] = {X 392.1701, Y 91.1451, Z -1.3333, A 0.000, B 0.000, C 0.000 }
gfCNCPoint1[6796] = {X 393.2723, Y 90.4949, Z -1.3333, A 0.000, B 0.000, C 0.000 }
gfCNCPoint1[6797] = {X 394.4714, Y 90.0477, Z -1.3333, A 0.000, B 0.000, C 0.000 }
gfCNCPoint1[6798] = {X 395.4063, Y 89.8549, Z -1.3333, A 0.000, B 0.000, C 0.000 }
gfCNCPoint1[6799] = {X 396.3584, Y 89.7861, Z -1.3333, A 0.000, B 0.000, C 0.000 }
gfCNCPoint1[6800] = {X 397.1501, Y 89.7496, Z -1.3333, A 0.000, B 0.000, C 0.000 }
gfCNCPoint1[6801] = {X 397.9389, Y 89.6717, Z -1.3333, A 0.000, B 0.000, C 0.000 }
gfCNCPoint1[6802] = {X 421.5726, Y 74.5352, Z -1.3333, A 0.000, B 0.000, C 0.000 }
gfCNCPoint1[6803] = {X 402.6720, Y 67.1191, Z -1.3333, A 0.000, B 0.000, C 0.000 }
gfCNCPoint1[6804] = {X 401.3008, Y 66.6641, Z -1.3333, A 0.000, B 0.000, C 0.000 }
gfCNCPoint1[6805] = {X 399.8883, Y 66.3610, Z -1.3333, A 0.000, B 0.000, C 0.000 }
gfCNCPoint1[6806] = {X 398.4511, Y 66.2133, Z -1.3333, A 0.000, B 0.000, C 0.000 }
gfCNCPoint1[6807] = {X 397.3064, Y 66.1057, Z -1.3333, A 0.000, B 0.000, C 0.000 }
gfCNCPoint1[6808] = {X 396.1929, Y 65.8193, Z -1.3333, A 0.000, B 0.000, C 0.000 }
gfCNCPoint1[6809] = {X 395.1383, Y 65.3611, Z -1.3333, A 0.000, B 0.000, C 0.000 }
gfCNCPoint1[6810] = {X 394.1691, Y 64.7425, Z -1.3333, A 0.000, B 0.000, C 0.000 }
gfCNCPoint1[6811] = {X 393.3093, Y 63.9791, Z -1.3333, A 0.000, B 0.000, C 0.000 }
gfCNCPoint1[6812] = {X 392.5117, Y 64.6967, Z -1.3333, A 0.000, B 0.000, C 0.000 }
gfCNCPoint1[6813] = {X 391.6175, Y 65.2895, Z -1.3333, A 0.000, B 0.000, C 0.000 }
gfCNCPoint1[6814] = {X 391.6167, Y 73.4805, Z -1.3333, A 0.000, B 0.000, C 0.000 }
gfCNCPoint1[6815] = {X 389.2167, Y 73.4803, Z -1.3333, A 0.000, B 0.000, C 0.000 }
gfCNCPoint1[6816] = {X 389.2156, Y 84.6139, Z -1.3333, A 0.000, B 0.000, C 0.000 }
gfCNCPoint1[6817] = {X 389.1536, Y 86.3199, Z -1.3333, A 0.000, B 0.000, C 0.000 }
gfCNCPoint1[6818] = {X 388.9432, Y 88.0140, Z -1.3333, A 0.000, B 0.000, C 0.000 }
gfCNCPoint1[6819] = {X 388.5862, Y 89.6833, Z -1.3333, A 0.000, B 0.000, C 0.000 }
gfCNCPoint1[6820] = {X 388.1032, Y 91.1629, Z -1.3333, A 0.000, B 0.000, C 0.000 }
gfCNCPoint1[6821] = {X 387.4395, Y 92.5707, Z -1.3333, A 0.000, B 0.000, C 0.000 }
gfCNCPoint1[6822] = {X 386.6055, Y 93.8848, Z -1.3333, A 0.000, B 0.000, C 0.000 }
gfCNCPoint1[6823] = {X 385.8731, Y 94.7997, Z -1.3333, A 0.000, B 0.000, C 0.000 }
gfCNCPoint1[6824] = {X 385.0581, Y 95.6418, Z -1.3333, A 0.000, B 0.000, C 0.000 }
gfCNCPoint1[6825] = {X 383.7979, Y 96.7248, Z -1.3333, A 0.000, B 0.000, C 0.000 }
gfCNCPoint1[6826] = {X 382.4487, Y 97.6949, Z -1.3333, A 0.000, B 0.000, C 0.000 }
gfCNCPoint1[6827] = {X 382.1856, Y 97.2934, Z -1.3333, A 0.000, B 0.000, C 0.000 }
gfCNCPoint1[6828] = {X 381.0191, Y 97.9984, Z -1.3333, A 0.000, B 0.000, C 0.000 }
gfCNCPoint1[6829] = {X 379.8043, Y 98.6167, Z -1.3333, A 0.000, B 0.000, C 0.000 }
gfCNCPoint1[6830] = {X 377.5277, Y 99.5764, Z -1.3333, A 0.000, B 0.000, C 0.000 }
gfCNCPoint1[6831] = {X 375.1876, Y 100.3686, Z -1.3333, A 0.000, B 0.000, C 0.000 }
gfCNCPoint1[6832] = {X 372.7962, Y 100.9893, Z -1.3333, A 0.000, B 0.000, C 0.000 }
gfCNCPoint1[6833] = {X 368.9811, Y 101.7274, Z -1.3333, A 0.000, B 0.000, C 0.000 }
gfCNCPoint1[6834] = {X 365.1349, Y 102.2812, Z -1.3333, A 0.000, B 0.000, C 0.000 }
gfCNCPoint1[6835] = {X 361.2665, Y 102.6495, Z -1.3333, A 0.000, B 0.000, C 0.000 }
gfCNCPoint1[6836] = {X 355.1239, Y 102.9828, Z -1.3333, A 0.000, B 0.000, C 0.000 }
gfCNCPoint1[6837] = {X 348.9737, Y 103.1113, Z -1.3333, A 0.000, B 0.000, C 0.000 }
gfCNCPoint1[6838] = {X 342.8225, Y 103.0349, Z -1.3333, A 0.000, B 0.000, C 0.000 }
gfCNCPoint1[6839] = {X 336.6774, Y 102.7536, Z -1.3333, A 0.000, B 0.000, C 0.000 }
gfCNCPoint1[6840] = {X 333.1844, Y 102.4784, Z -1.3333, A 0.000, B 0.000, C 0.000 }
gfCNCPoint1[6841] = {X 329.7050, Y 102.0651, Z -1.3333, A 0.000, B 0.000, C 0.000 }
gfCNCPoint1[6842] = {X 326.2448, Y 101.5144, Z -1.3333, A 0.000, B 0.000, C 0.000 }
gfCNCPoint1[6843] = {X 323.3896, Y 100.9088, Z -1.3333, A 0.000, B 0.000, C 0.000 }
gfCNCPoint1[6844] = {X 320.5869, Y 100.0942, Z -1.3333, A 0.000, B 0.000, C 0.000 }
gfCNCPoint1[6845] = {X 317.8519, Y 99.0753, Z -1.3333, A 0.000, B 0.000, C 0.000 }
gfCNCPoint1[6846] = {X 316.3326, Y 98.3753, Z -1.3333, A 0.000, B 0.000, C 0.000 }
gfCNCPoint1[6847] = {X 314.8774, Y 97.5504, Z -1.3333, A 0.000, B 0.000, C 0.000 }
gfCNCPoint1[6848] = {X 313.4965, Y 96.6062, Z -1.3333, A 0.000, B 0.000, C 0.000 }
gfCNCPoint1[6849] = {X 312.1996, Y 95.5496, Z -1.3333, A 0.000, B 0.000, C 0.000 }
gfCNCPoint1[6850] = {X 311.1896, Y 94.5444, Z -1.3333, A 0.000, B 0.000, C 0.000 }
gfCNCPoint1[6851] = {X 310.3058, Y 93.4266, Z -1.3333, A 0.000, B 0.000, C 0.000 }
gfCNCPoint1[6852] = {X 309.5607, Y 92.2119, Z -1.3333, A 0.000, B 0.000, C 0.000 }
gfCNCPoint1[6853] = {X 308.9647, Y 90.9175, Z -1.3333, A 0.000, B 0.000, C 0.000 }
gfCNCPoint1[6854] = {X 308.5263, Y 89.5616, Z -1.3333, A 0.000, B 0.000, C 0.000 }
gfCNCPoint1[6855] = {X 308.1815, Y 87.9321, Z -1.3333, A 0.000, B 0.000, C 0.000 }
gfCNCPoint1[6856] = {X 307.9778, Y 86.2789, Z -1.3333, A 0.000, B 0.000, C 0.000 }
gfCNCPoint1[6857] = {X 307.9167, Y 84.6144, Z -1.3333, A 0.000, B 0.000, C 0.000 }
gfCNCPoint1[6858] = {X 307.9180, Y 83.2309, Z -1.3333, A 0.000, B 0.000, C 0.000 }
gfCNCPoint1[6859] = {X 307.9180, Y 63.2815, Z -1.3333, A 0.000, B 0.000, C 0.000 }
gfCNCPoint1[6860] = {X 307.0584, Y 63.0566, Z -1.3333, A 0.000, B 0.000, C 0.000 }
gfCNCPoint1[6861] = {X 306.2614, Y 62.6635, Z -1.3333, A 0.000, B 0.000, C 0.000 }
gfCNCPoint1[6862] = {X 305.5598, Y 62.1184, Z -1.3333, A 0.000, B 0.000, C 0.000 }
gfCNCPoint1[6863] = {X 304.9819, Y 61.4434, Z -1.3333, A 0.000, B 0.000, C 0.000 }
gfCNCPoint1[6864] = {X 304.5514, Y 60.6660, Z -1.3333, A 0.000, B 0.000, C 0.000 }
gfCNCPoint1[6865] = {X 304.2859, Y 59.8181, Z -1.3333, A 0.000, B 0.000, C 0.000 }
gfCNCPoint1[6866] = {X 304.1962, Y 58.9340, Z -1.3333, A 0.000, B 0.000, C 0.000 }
gfCNCPoint1[6867] = {X 304.1962, Y 58.0000, Z -1.3333, A 0.000, B 0.000, C 0.000 }
gfCNCPoint1[6868] = {X 304.3065, Y 57.0209, Z -1.3333, A 0.000, B 0.000, C 0.000 }
gfCNCPoint1[6869] = {X 304.6320, Y 56.0909, Z -1.3333, A 0.000, B 0.000, C 0.000 }
gfCNCPoint1[6870] = {X 305.1562, Y 55.2566, Z -1.3333, A 0.000, B 0.000, C 0.000 }
gfCNCPoint1[6871] = {X 305.8529, Y 54.5599, Z -1.3333, A 0.000, B 0.000, C 0.000 }
gfCNCPoint1[6872] = {X 306.6871, Y 54.0357, Z -1.3333, A 0.000, B 0.000, C 0.000 }
gfCNCPoint1[6873] = {X 307.6171, Y 53.7103, Z -1.3333, A 0.000, B 0.000, C 0.000 }
gfCNCPoint1[6874] = {X 308.5962, Y 53.6000, Z -1.3333, A 0.000, B 0.000, C 0.000 }
gfCNCPoint1[6875] = {X 324.3107, Y 53.6000, Z -1.3333, A 0.000, B 0.000, C 0.000 }
gfCNCPoint1[6876] = {X 325.2898, Y 53.7103, Z -1.3333, A 0.000, B 0.000, C 0.000 }
gfCNCPoint1[6877] = {X 326.2198, Y 54.0357, Z -1.3333, A 0.000, B 0.000, C 0.000 }
gfCNCPoint1[6878] = {X 327.0540, Y 54.5599, Z -1.3333, A 0.000, B 0.000, C 0.000 }
gfCNCPoint1[6879] = {X 327.7507, Y 55.2566, Z -1.3333, A 0.000, B 0.000, C 0.000 }
gfCNCPoint1[6880] = {X 328.2750, Y 56.0909, Z -1.3333, A 0.000, B 0.000, C 0.000 }
gfCNCPoint1[6881] = {X 328.6004, Y 57.0209, Z -1.3333, A 0.000, B 0.000, C 0.000 }
gfCNCPoint1[6882] = {X 328.7107, Y 58.0000, Z -1.3333, A 0.000, B 0.000, C 0.000 }
gfCNCPoint1[6883] = {X 328.7107, Y 58.9366, Z -1.3333, A 0.000, B 0.000, C 0.000 }
gfCNCPoint1[6884] = {X 328.6164, Y 59.8192, Z -1.3333, A 0.000, B 0.000, C 0.000 }
gfCNCPoint1[6885] = {X 328.3485, Y 60.6653, Z -1.3333, A 0.000, B 0.000, C 0.000 }
gfCNCPoint1[6886] = {X 327.9176, Y 61.4413, Z -1.3333, A 0.000, B 0.000, C 0.000 }
gfCNCPoint1[6887] = {X 327.3410, Y 62.1160, Z -1.3333, A 0.000, B 0.000, C 0.000 }
gfCNCPoint1[6888] = {X 326.6417, Y 62.6626, Z -1.3333, A 0.000, B 0.000, C 0.000 }
gfCNCPoint1[6889] = {X 325.8476, Y 63.0592, Z -1.3333, A 0.000, B 0.000, C 0.000 }
gfCNCPoint1[6890] = {X 324.9906, Y 63.2899, Z -1.3333, A 0.000, B 0.000, C 0.000 }
gfCNCPoint1[6891] = {X 324.9919, Y 83.2292, Z -1.3333, A 0.000, B 0.000, C 0.000 }
gfCNCPoint1[6892] = {X 325.0054, Y 84.6147, Z -1.3333, A 0.000, B 0.000, C 0.000 }
gfCNCPoint1[6893] = {X 325.0812, Y 85.8328, Z -1.3333, A 0.000, B 0.000, C 0.000 }
gfCNCPoint1[6894] = {X 325.3000, Y 87.0336, Z -1.3333, A 0.000, B 0.000, C 0.000 }
gfCNCPoint1[6895] = {X 325.5330, Y 87.2845, Z -1.3333, A 0.000, B 0.000, C 0.000 }
gfCNCPoint1[6896] = {X 325.8184, Y 87.4736, Z -1.3333, A 0.000, B 0.000, C 0.000 }
gfCNCPoint1[6897] = {X 326.2603, Y 87.7228, Z -1.3333, A 0.000, B 0.000, C 0.000 }
gfCNCPoint1[6898] = {X 327.6903, Y 88.3168, Z -1.3333, A 0.000, B 0.000, C 0.000 }
gfCNCPoint1[6899] = {X 329.1770, Y 88.7499, Z -1.3333, A 0.000, B 0.000, C 0.000 }
gfCNCPoint1[6900] = {X 332.2480, Y 89.3646, Z -1.3333, A 0.000, B 0.000, C 0.000 }
gfCNCPoint1[6901] = {X 335.3554, Y 89.7561, Z -1.3333, A 0.000, B 0.000, C 0.000 }
gfCNCPoint1[6902] = {X 340.5274, Y 90.1388, Z -1.3333, A 0.000, B 0.000, C 0.000 }
gfCNCPoint1[6903] = {X 345.7116, Y 90.2833, Z -1.3333, A 0.000, B 0.000, C 0.000 }
gfCNCPoint1[6904] = {X 350.5506, Y 90.2892, Z -1.3333, A 0.000, B 0.000, C 0.000 }
gfCNCPoint1[6905] = {X 355.3867, Y 90.1207, Z -1.3333, A 0.000, B 0.000, C 0.000 }
gfCNCPoint1[6906] = {X 360.2136, Y 89.7781, Z -1.3333, A 0.000, B 0.000, C 0.000 }
gfCNCPoint1[6907] = {X 362.7550, Y 89.4894, Z -1.3333, A 0.000, B 0.000, C 0.000 }
gfCNCPoint1[6908] = {X 365.2730, Y 89.0401, Z -1.3333, A 0.000, B 0.000, C 0.000 }
gfCNCPoint1[6909] = {X 367.7574, Y 88.4322, Z -1.3333, A 0.000, B 0.000, C 0.000 }
gfCNCPoint1[6910] = {X 368.6805, Y 88.1217, Z -1.3333, A 0.000, B 0.000, C 0.000 }
gfCNCPoint1[6911] = {X 369.5630, Y 87.7096, Z -1.3333, A 0.000, B 0.000, C 0.000 }
gfCNCPoint1[6912] = {X 370.3937, Y 87.2012, Z -1.3333, A 0.000, B 0.000, C 0.000 }
gfCNCPoint1[6913] = {X 370.5217, Y 87.0680, Z -1.3333, A 0.000, B 0.000, C 0.000 }
gfCNCPoint1[6914] = {X 370.5877, Y 86.8954, Z -1.3333, A 0.000, B 0.000, C 0.000 }
gfCNCPoint1[6915] = {X 370.7779, Y 85.3668, Z -1.3333, A 0.000, B 0.000, C 0.000 }
gfCNCPoint1[6916] = {X 370.8414, Y 83.8276, Z -1.3333, A 0.000, B 0.000, C 0.000 }
gfCNCPoint1[6917] = {X 370.8397, Y 63.2813, Z -1.3333, A 0.000, B 0.000, C 0.000 }
gfCNCPoint1[6918] = {X 369.9803, Y 63.0561, Z -1.3333, A 0.000, B 0.000, C 0.000 }
gfCNCPoint1[6919] = {X 369.1837, Y 62.6630, Z -1.3333, A 0.000, B 0.000, C 0.000 }
gfCNCPoint1[6920] = {X 368.4822, Y 62.1178, Z -1.3333, A 0.000, B 0.000, C 0.000 }
gfCNCPoint1[6921] = {X 367.9046, Y 61.4429, Z -1.3333, A 0.000, B 0.000, C 0.000 }
gfCNCPoint1[6922] = {X 367.4743, Y 60.6657, Z -1.3333, A 0.000, B 0.000, C 0.000 }
gfCNCPoint1[6923] = {X 367.2090, Y 59.8179, Z -1.3333, A 0.000, B 0.000, C 0.000 }
gfCNCPoint1[6924] = {X 367.1193, Y 58.9340, Z -1.3333, A 0.000, B 0.000, C 0.000 }
gfCNCPoint1[6925] = {X 367.1193, Y 58.0000, Z -1.3333, A 0.000, B 0.000, C 0.000 }
gfCNCPoint1[6926] = {X 367.2296, Y 57.0209, Z -1.3333, A 0.000, B 0.000, C 0.000 }
gfCNCPoint1[6927] = {X 367.5550, Y 56.0909, Z -1.3333, A 0.000, B 0.000, C 0.000 }
gfCNCPoint1[6928] = {X 368.0792, Y 55.2566, Z -1.3333, A 0.000, B 0.000, C 0.000 }
gfCNCPoint1[6929] = {X 368.7759, Y 54.5599, Z -1.3333, A 0.000, B 0.000, C 0.000 }
gfCNCPoint1[6930] = {X 369.6102, Y 54.0357, Z -1.3333, A 0.000, B 0.000, C 0.000 }
gfCNCPoint1[6931] = {X 370.5402, Y 53.7103, Z -1.3333, A 0.000, B 0.000, C 0.000 }
gfCNCPoint1[6932] = {X 371.5193, Y 53.6000, Z -1.3333, A 0.000, B 0.000, C 0.000 }
gfCNCPoint1[6933] = {X 388.0597, Y 53.6000, Z -1.3333, A 0.000, B 0.000, C 0.000 }
gfCNCPoint1[6934] = {X 389.0388, Y 53.7103, Z -1.3333, A 0.000, B 0.000, C 0.000 }
gfCNCPoint1[6935] = {X 389.9688, Y 54.0357, Z -1.3333, A 0.000, B 0.000, C 0.000 }
gfCNCPoint1[6936] = {X 390.8030, Y 54.5599, Z -1.3333, A 0.000, B 0.000, C 0.000 }
gfCNCPoint1[6937] = {X 391.4997, Y 55.2566, Z -1.3333, A 0.000, B 0.000, C 0.000 }
gfCNCPoint1[6938] = {X 392.0239, Y 56.0909, Z -1.3333, A 0.000, B 0.000, C 0.000 }
gfCNCPoint1[6939] = {X 392.3494, Y 57.0209, Z -1.3333, A 0.000, B 0.000, C 0.000 }
gfCNCPoint1[6940] = {X 392.4597, Y 58.0000, Z -1.3333, A 0.000, B 0.000, C 0.000 }
gfCNCPoint1[6941] = {X 392.4595, Y 58.9704, Z -1.3333, A 0.000, B 0.000, C 0.000 }
gfCNCPoint1[6942] = {X 392.3370, Y 59.9657, Z -1.3333, A 0.000, B 0.000, C 0.000 }
gfCNCPoint1[6943] = {X 391.9924, Y 60.9074, Z -1.3333, A 0.000, B 0.000, C 0.000 }
gfCNCPoint1[6944] = {X 391.5482, Y 61.6162, Z -1.3333, A 0.000, B 0.000, C 0.000 }
gfCNCPoint1[6945] = {X 390.9784, Y 62.2286, Z -1.3333, A 0.000, B 0.000, C 0.000 }
gfCNCPoint1[6946] = {X 390.3034, Y 62.7227, Z -1.3333, A 0.000, B 0.000, C 0.000 }
gfCNCPoint1[6947] = {X 389.5475, Y 63.0809, Z -1.3333, A 0.000, B 0.000, C 0.000 }
gfCNCPoint1[6948] = {X 388.7376, Y 63.2902, Z -1.3333, A 0.000, B 0.000, C 0.000 }
gfCNCPoint1[6949] = {X 388.7376, Y 83.9247, Z -1.3333, A 0.000, B 0.000, C 0.000 }
gfCNCPoint1[6950] = {X 388.7356, Y 84.6150, Z -1.3333, A 0.000, B 0.000, C 0.000 }
gfCNCPoint1[6951] = {X 388.6753, Y 86.2800, Z -1.3333, A 0.000, B 0.000, C 0.000 }
gfCNCPoint1[6952] = {X 388.4701, Y 87.9333, Z -1.3333, A 0.000, B 0.000, C 0.000 }
gfCNCPoint1[6953] = {X 388.1216, Y 89.5626, Z -1.3333, A 0.000, B 0.000, C 0.000 }
gfCNCPoint1[6954] = {X 387.5859, Y 91.1607, Z -1.3333, A 0.000, B 0.000, C 0.000 }
gfCNCPoint1[6955] = {X 386.8313, Y 92.6679, Z -1.3333, A 0.000, B 0.000, C 0.000 }
gfCNCPoint1[6956] = {X 385.8726, Y 94.0543, Z -1.3333, A 0.000, B 0.000, C 0.000 }
gfCNCPoint1[6957] = {X 384.7288, Y 95.2925, Z -1.3333, A 0.000, B 0.000, C 0.000 }
gfCNCPoint1[6958] = {X 383.5005, Y 96.3480, Z -1.3333, A 0.000, B 0.000, C 0.000 }
gfCNCPoint1[6959] = {X 382.1856, Y 97.2934, Z -1.3333, A 0.000, B 0.000, C 0.000 }
gfCNCPoint1[6960] = {X 382.4487, Y 97.6949, Z -1.3333, A 0.000, B 0.000, C 0.000 }
gfCNCPoint1[6961] = {X 391.5260, Y 97.6949, Z -1.3333, A 0.000, B 0.000, C 0.000 }
gfCNCPoint1[6962] = {X 391.5260, Y 97.0659, Z -1.3333, A 0.000, B 0.000, C 0.000 }
gfCNCPoint1[6963] = {X 391.6192, Y 96.1165, Z -1.3333, A 0.000, B 0.000, C 0.000 }
gfCNCPoint1[6964] = {X 391.8954, Y 95.2034, Z -1.3333, A 0.000, B 0.000, C 0.000 }
gfCNCPoint1[6965] = {X 392.3440, Y 94.3614, Z -1.3333, A 0.000, B 0.000, C 0.000 }
gfCNCPoint1[6966] = {X 392.9478, Y 93.6228, Z -1.3333, A 0.000, B 0.000, C 0.000 }
gfCNCPoint1[6967] = {X 393.6837, Y 93.0158, Z -1.3333, A 0.000, B 0.000, C 0.000 }
gfCNCPoint1[6968] = {X 394.5237, Y 92.5635, Z -1.3333, A 0.000, B 0.000, C 0.000 }
gfCNCPoint1[6969] = {X 395.4357, Y 92.2834, Z -1.3333, A 0.000, B 0.000, C 0.000 }
gfCNCPoint1[6970] = {X 396.3847, Y 92.1860, Z -1.3333, A 0.000, B 0.000, C 0.000 }
gfCNCPoint1[6971] = {X 397.3063, Y 92.1471, Z -1.3333, A 0.000, B 0.000, C 0.000 }
gfCNCPoint1[6972] = {X 398.2246, Y 92.0599, Z -1.3333, A 0.000, B 0.000, C 0.000 }
gfCNCPoint1[6973] = {X 398.7527, Y 91.9318, Z -1.3333, A 0.000, B 0.000, C 0.000 }
gfCNCPoint1[6974] = {X 399.2389, Y 91.6891, Z -1.3333, A 0.000, B 0.000, C 0.000 }
gfCNCPoint1[6975] = {X 426.8282, Y 74.0193, Z -1.3333, A 0.000, B 0.000, C 0.000 }
gfCNCPoint1[6976] = {X 403.5508, Y 64.8858, Z -1.3333, A 0.000, B 0.000, C 0.000 }
gfCNCPoint1[6977] = {X 401.9168, Y 64.3445, Z -1.3333, A 0.000, B 0.000, C 0.000 }
gfCNCPoint1[6978] = {X 400.2333, Y 63.9857, Z -1.3333, A 0.000, B 0.000, C 0.000 }
gfCNCPoint1[6979] = {X 398.5206, Y 63.8139, Z -1.3333, A 0.000, B 0.000, C 0.000 }
gfCNCPoint1[6980] = {X 397.5548, Y 63.7099, Z -1.3333, A 0.000, B 0.000, C 0.000 }
gfCNCPoint1[6981] = {X 396.6287, Y 63.4166, Z -1.3333, A 0.000, B 0.000, C 0.000 }
gfCNCPoint1[6982] = {X 395.7791, Y 62.9458, Z -1.3333, A 0.000, B 0.000, C 0.000 }
gfCNCPoint1[6983] = {X 395.0396, Y 62.3159, Z -1.3333, A 0.000, B 0.000, C 0.000 }
gfCNCPoint1[6984] = {X 394.4659, Y 61.5933, Z -1.3333, A 0.000, B 0.000, C 0.000 }
gfCNCPoint1[6985] = {X 394.0385, Y 60.7756, Z -1.3333, A 0.000, B 0.000, C 0.000 }
gfCNCPoint1[6986] = {X 393.7727, Y 59.8921, Z -1.3333, A 0.000, B 0.000, C 0.000 }
gfCNCPoint1[6987] = {X 393.6779, Y 58.9744, Z -1.3333, A 0.000, B 0.000, C 0.000 }
gfCNCPoint1[6988] = {X 393.6777, Y 58.0000, Z -1.3333, A 0.000, B 0.000, C 0.000 }
gfCNCPoint1[6989] = {X 393.7668, Y 57.0718, Z -1.3333, A 0.000, B 0.000, C 0.000 }
gfCNCPoint1[6990] = {X 394.0309, Y 56.1774, Z -1.3333, A 0.000, B 0.000, C 0.000 }
gfCNCPoint1[6991] = {X 394.4602, Y 55.3496, Z -1.3333, A 0.000, B 0.000, C 0.000 }
gfCNCPoint1[6992] = {X 395.0391, Y 54.6186, Z -1.3333, A 0.000, B 0.000, C 0.000 }
gfCNCPoint1[6993] = {X 395.7864, Y 53.9833, Z -1.3333, A 0.000, B 0.000, C 0.000 }
gfCNCPoint1[6994] = {X 396.6455, Y 53.5102, Z -1.3333, A 0.000, B 0.000, C 0.000 }
gfCNCPoint1[6995] = {X 397.5819, Y 53.2186, Z -1.3333, A 0.000, B 0.000, C 0.000 }
gfCNCPoint1[6996] = {X 398.5577, Y 53.1200, Z -1.3333, A 0.000, B 0.000, C 0.000 }
gfCNCPoint1[6997] = {X 419.4886, Y 53.1200, Z -1.3333, A 0.000, B 0.000, C 0.000 }
gfCNCPoint1[6998] = {X 420.5535, Y 53.2376, Z -1.3333, A 0.000, B 0.000, C 0.000 }
gfCNCPoint1[6999] = {X 421.5671, Y 53.5848, Z -1.3333, A 0.000, B 0.000, C 0.000 }
gfCNCPoint1[7000] = {X 422.4804, Y 54.1447, Z -1.3333, A 0.000, B 0.000, C 0.000 }
gfCNCPoint1[7001] = {X 423.2496, Y 54.8905, Z -1.3333, A 0.000, B 0.000, C 0.000 }
gfCNCPoint1[7002] = {X 423.8375, Y 55.7861, Z -1.3333, A 0.000, B 0.000, C 0.000 }
gfCNCPoint1[7003] = {X 424.2158, Y 56.7885, Z -1.3333, A 0.000, B 0.000, C 0.000 }
gfCNCPoint1[7004] = {X 424.3663, Y 57.8492, Z -1.3333, A 0.000, B 0.000, C 0.000 }
gfCNCPoint1[7005] = {X 429.8190, Y 59.9745, Z -1.3333, A 0.000, B 0.000, C 0.000 }
gfCNCPoint1[7006] = {X 457.3013, Y 70.8779, Z -1.3333, A 0.000, B 0.000, C 0.000 }
gfCNCPoint1[7007] = {X 457.3001, Y 63.6743, Z -1.3333, A 0.000, B 0.000, C 0.000 }
gfCNCPoint1[7008] = {X 456.2917, Y 63.3061, Z -1.3333, A 0.000, B 0.000, C 0.000 }
gfCNCPoint1[7009] = {X 455.3882, Y 62.7263, Z -1.3333, A 0.000, B 0.000, C 0.000 }
gfCNCPoint1[7010] = {X 454.6333, Y 61.9629, Z -1.3333, A 0.000, B 0.000, C 0.000 }
gfCNCPoint1[7011] = {X 454.0636, Y 61.0529, Z -1.3333, A 0.000, B 0.000, C 0.000 }
gfCNCPoint1[7012] = {X 453.7067, Y 60.0404, Z -1.3333, A 0.000, B 0.000, C 0.000 }
gfCNCPoint1[7013] = {X 453.5798, Y 58.9744, Z -1.3333, A 0.000, B 0.000, C 0.000 }
gfCNCPoint1[7014] = {X 453.5796, Y 58.0000, Z -1.3333, A 0.000, B 0.000, C 0.000 }
gfCNCPoint1[7015] = {X 453.6734, Y 57.0480, Z -1.3333, A 0.000, B 0.000, C 0.000 }
gfCNCPoint1[7016] = {X 453.9511, Y 56.1325, Z -1.3333, A 0.000, B 0.000, C 0.000 }
gfCNCPoint1[7017] = {X 454.4020, Y 55.2888, Z -1.3333, A 0.000, B 0.000, C 0.000 }
gfCNCPoint1[7018] = {X 455.0089, Y 54.5493, Z -1.3333, A 0.000, B 0.000, C 0.000 }
gfCNCPoint1[7019] = {X 455.7484, Y 53.9424, Z -1.3333, A 0.000, B 0.000, C 0.000 }
gfCNCPoint1[7020] = {X 456.5921, Y 53.4915, Z -1.3333, A 0.000, B 0.000, C 0.000 }
gfCNCPoint1[7021] = {X 457.5076, Y 53.2138, Z -1.3333, A 0.000, B 0.000, C 0.000 }
gfCNCPoint1[7022] = {X 458.4596, Y 53.1200, Z -1.3333, A 0.000, B 0.000, C 0.000 }
gfCNCPoint1[7023] = {X 475.0000, Y 53.1200, Z -1.3333, A 0.000, B 0.000, C 0.000 }
gfCNCPoint1[7024] = {X 475.9520, Y 53.2138, Z -1.3333, A 0.000, B 0.000, C 0.000 }
gfCNCPoint1[7025] = {X 476.8675, Y 53.4915, Z -1.3333, A 0.000, B 0.000, C 0.000 }
gfCNCPoint1[7026] = {X 477.7112, Y 53.9424, Z -1.3333, A 0.000, B 0.000, C 0.000 }
gfCNCPoint1[7027] = {X 478.4507, Y 54.5493, Z -1.3333, A 0.000, B 0.000, C 0.000 }
gfCNCPoint1[7028] = {X 479.0576, Y 55.2888, Z -1.3333, A 0.000, B 0.000, C 0.000 }
gfCNCPoint1[7029] = {X 479.5085, Y 56.1325, Z -1.3333, A 0.000, B 0.000, C 0.000 }
gfCNCPoint1[7030] = {X 479.7862, Y 57.0480, Z -1.3333, A 0.000, B 0.000, C 0.000 }
gfCNCPoint1[7031] = {X 479.8800, Y 58.0000, Z -1.3333, A 0.000, B 0.000, C 0.000 }
gfCNCPoint1[7032] = {X 479.8798, Y 58.9744, Z -1.3333, A 0.000, B 0.000, C 0.000 }
gfCNCPoint1[7033] = {X 479.7529, Y 60.0405, Z -1.3333, A 0.000, B 0.000, C 0.000 }
gfCNCPoint1[7034] = {X 479.3960, Y 61.0530, Z -1.3333, A 0.000, B 0.000, C 0.000 }
gfCNCPoint1[7035] = {X 478.8262, Y 61.9630, Z -1.3333, A 0.000, B 0.000, C 0.000 }
gfCNCPoint1[7036] = {X 478.0713, Y 62.7264, Z -1.3333, A 0.000, B 0.000, C 0.000 }
gfCNCPoint1[7037] = {X 477.1677, Y 63.3062, Z -1.3333, A 0.000, B 0.000, C 0.000 }
gfCNCPoint1[7038] = {X 476.1592, Y 63.6744, Z -1.3333, A 0.000, B 0.000, C 0.000 }
gfCNCPoint1[7039] = {X 476.1596, Y 92.3325, Z -1.3333, A 0.000, B 0.000, C 0.000 }
gfCNCPoint1[7040] = {X 476.3622, Y 92.3919, Z -1.3333, A 0.000, B 0.000, C 0.000 }
gfCNCPoint1[7041] = {X 476.5632, Y 92.4562, Z -1.3333, A 0.000, B 0.000, C 0.000 }
gfCNCPoint1[7042] = {X 477.4813, Y 92.8732, Z -1.3333, A 0.000, B 0.000, C 0.000 }
gfCNCPoint1[7043] = {X 478.2933, Y 93.4708, Z -1.3333, A 0.000, B 0.000, C 0.000 }
gfCNCPoint1[7044] = {X 478.9645, Y 94.2233, Z -1.3333, A 0.000, B 0.000, C 0.000 }
gfCNCPoint1[7045] = {X 479.4657, Y 95.0982, Z -1.3333, A 0.000, B 0.000, C 0.000 }
gfCNCPoint1[7046] = {X 479.7753, Y 96.0577, Z -1.3333, A 0.000, B 0.000, C 0.000 }
gfCNCPoint1[7047] = {X 479.8800, Y 97.0605, Z -1.3333, A 0.000, B 0.000, C 0.000 }
gfCNCPoint1[7048] = {X 479.8800, Y 97.6949, Z -1.3333, A 0.000, B 0.000, C 0.000 }
gfCNCPoint1[7049] = {X 479.4000, Y 97.6949, Z -1.3333, A 0.000, B 0.000, C 0.000 }
gfCNCPoint1[7050] = {X 479.4000, Y 98.0000, Z -1.3333, A 0.000, B 0.000, C 0.000 }
gfCNCPoint1[7051] = {X 479.2897, Y 98.9791, Z -1.3333, A 0.000, B 0.000, C 0.000 }
gfCNCPoint1[7052] = {X 478.9643, Y 99.9091, Z -1.3333, A 0.000, B 0.000, C 0.000 }
gfCNCPoint1[7053] = {X 478.4401, Y 100.7434, Z -1.3333, A 0.000, B 0.000, C 0.000 }
gfCNCPoint1[7054] = {X 477.7434, Y 101.4401, Z -1.3333, A 0.000, B 0.000, C 0.000 }
gfCNCPoint1[7055] = {X 476.9091, Y 101.9643, Z -1.3333, A 0.000, B 0.000, C 0.000 }
gfCNCPoint1[7056] = {X 475.9791, Y 102.2897, Z -1.3333, A 0.000, B 0.000, C 0.000 }
gfCNCPoint1[7057] = {X 475.0000, Y 102.4000, Z -1.3333, A 0.000, B 0.000, C 0.000 }
gfCNCPoint1[7058] = {X 458.4596, Y 102.4000, Z -1.3333, A 0.000, B 0.000, C 0.000 }
gfCNCPoint1[7059] = {X 457.4805, Y 102.2897, Z -1.3333, A 0.000, B 0.000, C 0.000 }
gfCNCPoint1[7060] = {X 456.5505, Y 101.9643, Z -1.3333, A 0.000, B 0.000, C 0.000 }
gfCNCPoint1[7061] = {X 455.7162, Y 101.4401, Z -1.3333, A 0.000, B 0.000, C 0.000 }
gfCNCPoint1[7062] = {X 455.0195, Y 100.7434, Z -1.3333, A 0.000, B 0.000, C 0.000 }
gfCNCPoint1[7063] = {X 454.4953, Y 99.9091, Z -1.3333, A 0.000, B 0.000, C 0.000 }
gfCNCPoint1[7064] = {X 454.1699, Y 98.9791, Z -1.3333, A 0.000, B 0.000, C 0.000 }
gfCNCPoint1[7065] = {X 454.0596, Y 98.0000, Z -1.3333, A 0.000, B 0.000, C 0.000 }
gfCNCPoint1[7066] = {X 454.0596, Y 97.0659, Z -1.3333, A 0.000, B 0.000, C 0.000 }
gfCNCPoint1[7067] = {X 454.1492, Y 96.1826, Z -1.3333, A 0.000, B 0.000, C 0.000 }
gfCNCPoint1[7068] = {X 454.4143, Y 95.3353, Z -1.3333, A 0.000, B 0.000, C 0.000 }
gfCNCPoint1[7069] = {X 454.8440, Y 94.5584, Z -1.3333, A 0.000, B 0.000, C 0.000 }
gfCNCPoint1[7070] = {X 455.4210, Y 93.8836, Z -1.3333, A 0.000, B 0.000, C 0.000 }
gfCNCPoint1[7071] = {X 456.1217, Y 93.3384, Z -1.3333, A 0.000, B 0.000, C 0.000 }
gfCNCPoint1[7072] = {X 456.9176, Y 92.9450, Z -1.3333, A 0.000, B 0.000, C 0.000 }
gfCNCPoint1[7073] = {X 457.7763, Y 92.7193, Z -1.3333, A 0.000, B 0.000, C 0.000 }
gfCNCPoint1[7074] = {X 457.7763, Y 85.6495, Z -1.3333, A 0.000, B 0.000, C 0.000 }
gfCNCPoint1[7075] = {X 444.8669, Y 80.5890, Z -1.3333, A 0.000, B 0.000, C 0.000 }
gfCNCPoint1[7076] = {X 420.1029, Y 96.6312, Z -1.3333, A 0.000, B 0.000, C 0.000 }
gfCNCPoint1[7077] = {X 420.1067, Y 97.0659, Z -1.3333, A 0.000, B 0.000, C 0.000 }
gfCNCPoint1[7078] = {X 420.1067, Y 98.0000, Z -1.3333, A 0.000, B 0.000, C 0.000 }
gfCNCPoint1[7079] = {X 419.9964, Y 98.9791, Z -1.3333, A 0.000, B 0.000, C 0.000 }
gfCNCPoint1[7080] = {X 419.6710, Y 99.9091, Z -1.3333, A 0.000, B 0.000, C 0.000 }
gfCNCPoint1[7081] = {X 419.1468, Y 100.7434, Z -1.3333, A 0.000, B 0.000, C 0.000 }
gfCNCPoint1[7082] = {X 418.4501, Y 101.4401, Z -1.3333, A 0.000, B 0.000, C 0.000 }
gfCNCPoint1[7083] = {X 417.6158, Y 101.9643, Z -1.3333, A 0.000, B 0.000, C 0.000 }
gfCNCPoint1[7084] = {X 416.6858, Y 102.2897, Z -1.3333, A 0.000, B 0.000, C 0.000 }
gfCNCPoint1[7085] = {X 415.7067, Y 102.4000, Z -1.3333, A 0.000, B 0.000, C 0.000 }
gfCNCPoint1[7086] = {X 396.4059, Y 102.4000, Z -1.3333, A 0.000, B 0.000, C 0.000 }
gfCNCPoint1[7087] = {X 395.4269, Y 102.2897, Z -1.3333, A 0.000, B 0.000, C 0.000 }
gfCNCPoint1[7088] = {X 394.4969, Y 101.9643, Z -1.3333, A 0.000, B 0.000, C 0.000 }
gfCNCPoint1[7089] = {X 393.6626, Y 101.4401, Z -1.3333, A 0.000, B 0.000, C 0.000 }
gfCNCPoint1[7090] = {X 392.9659, Y 100.7434, Z -1.3333, A 0.000, B 0.000, C 0.000 }
gfCNCPoint1[7091] = {X 392.4417, Y 99.9091, Z -1.3333, A 0.000, B 0.000, C 0.000 }
gfCNCPoint1[7092] = {X 392.1163, Y 98.9791, Z -1.3333, A 0.000, B 0.000, C 0.000 }
gfCNCPoint1[7093] = {X 392.0059, Y 98.0000, Z -1.3333, A 0.000, B 0.000, C 0.000 }
gfCNCPoint1[7094] = {X 392.0059, Y 97.0659, Z -1.3333, A 0.000, B 0.000, C 0.000 }
gfCNCPoint1[7095] = {X 392.1157, Y 96.0891, Z -1.3333, A 0.000, B 0.000, C 0.000 }
gfCNCPoint1[7096] = {X 392.4396, Y 95.1611, Z -1.3333, A 0.000, B 0.000, C 0.000 }
gfCNCPoint1[7097] = {X 392.9615, Y 94.3281, Z -1.3333, A 0.000, B 0.000, C 0.000 }
gfCNCPoint1[7098] = {X 393.6552, Y 93.6318, Z -1.3333, A 0.000, B 0.000, C 0.000 }
gfCNCPoint1[7099] = {X 394.4863, Y 93.1068, Z -1.3333, A 0.000, B 0.000, C 0.000 }
gfCNCPoint1[7100] = {X 395.4131, Y 92.7794, Z -1.3333, A 0.000, B 0.000, C 0.000 }
gfCNCPoint1[7101] = {X 396.3895, Y 92.6660, Z -1.3333, A 0.000, B 0.000, C 0.000 }
gfCNCPoint1[7102] = {X 397.3382, Y 92.6260, Z -1.3333, A 0.000, B 0.000, C 0.000 }
gfCNCPoint1[7103] = {X 398.2835, Y 92.5363, Z -1.3333, A 0.000, B 0.000, C 0.000 }
gfCNCPoint1[7104] = {X 398.9174, Y 92.3826, Z -1.3333, A 0.000, B 0.000, C 0.000 }
gfCNCPoint1[7105] = {X 399.5010, Y 92.0913, Z -1.3333, A 0.000, B 0.000, C 0.000 }
gfCNCPoint1[7106] = {X 405.1781, Y 88.4328, Z -1.3333, A 0.000, B 0.000, C 0.000 }
gfCNCPoint1[7107] = {X 427.8801, Y 73.9164, Z -1.3333, A 0.000, B 0.000, C 0.000 }
gfCNCPoint1[7108] = {X 403.7261, Y 64.4389, Z -1.3333, A 0.000, B 0.000, C 0.000 }
gfCNCPoint1[7109] = {X 402.0392, Y 63.8803, Z -1.3333, A 0.000, B 0.000, C 0.000 }
gfCNCPoint1[7110] = {X 400.3011, Y 63.5105, Z -1.3333, A 0.000, B 0.000, C 0.000 }
gfCNCPoint1[7111] = {X 398.5329, Y 63.3340, Z -1.3333, A 0.000, B 0.000, C 0.000 }
gfCNCPoint1[7112] = {X 397.5579, Y 63.2190, Z -1.3333, A 0.000, B 0.000, C 0.000 }
gfCNCPoint1[7113] = {X 396.6327, Y 62.8906, Z -1.3333, A 0.000, B 0.000, C 0.000 }
gfCNCPoint1[7114] = {X 395.8033, Y 62.3653, Z -1.3333, A 0.000, B 0.000, C 0.000 }
gfCNCPoint1[7115] = {X 395.1110, Y 61.6691, Z -1.3333, A 0.000, B 0.000, C 0.000 }
gfCNCPoint1[7116] = {X 394.5904, Y 60.8368, Z -1.3333, A 0.000, B 0.000, C 0.000 }
gfCNCPoint1[7117] = {X 394.2672, Y 59.9097, Z -1.3333, A 0.000, B 0.000, C 0.000 }
gfCNCPoint1[7118] = {X 394.1577, Y 58.9340, Z -1.3333, A 0.000, B 0.000, C 0.000 }
gfCNCPoint1[7119] = {X 394.1577, Y 58.0000, Z -1.3333, A 0.000, B 0.000, C 0.000 }
gfCNCPoint1[7120] = {X 394.2680, Y 57.0209, Z -1.3333, A 0.000, B 0.000, C 0.000 }
gfCNCPoint1[7121] = {X 394.5935, Y 56.0909, Z -1.3333, A 0.000, B 0.000, C 0.000 }
gfCNCPoint1[7122] = {X 395.1177, Y 55.2566, Z -1.3333, A 0.000, B 0.000, C 0.000 }
gfCNCPoint1[7123] = {X 395.8144, Y 54.5599, Z -1.3333, A 0.000, B 0.000, C 0.000 }
gfCNCPoint1[7124] = {X 396.6486, Y 54.0357, Z -1.3333, A 0.000, B 0.000, C 0.000 }
gfCNCPoint1[7125] = {X 397.5786, Y 53.7103, Z -1.3333, A 0.000, B 0.000, C 0.000 }
gfCNCPoint1[7126] = {X 398.5577, Y 53.6000, Z -1.3333, A 0.000, B 0.000, C 0.000 }
gfCNCPoint1[7127] = {X 419.4886, Y 53.6000, Z -1.3333, A 0.000, B 0.000, C 0.000 }
gfCNCPoint1[7128] = {X 420.4677, Y 53.7103, Z -1.3333, A 0.000, B 0.000, C 0.000 }
gfCNCPoint1[7129] = {X 421.3977, Y 54.0357, Z -1.3333, A 0.000, B 0.000, C 0.000 }
gfCNCPoint1[7130] = {X 422.2320, Y 54.5599, Z -1.3333, A 0.000, B 0.000, C 0.000 }
gfCNCPoint1[7131] = {X 422.9287, Y 55.2566, Z -1.3333, A 0.000, B 0.000, C 0.000 }
gfCNCPoint1[7132] = {X 423.4529, Y 56.0909, Z -1.3333, A 0.000, B 0.000, C 0.000 }
gfCNCPoint1[7133] = {X 423.7783, Y 57.0209, Z -1.3333, A 0.000, B 0.000, C 0.000 }
gfCNCPoint1[7134] = {X 423.8886, Y 58.0000, Z -1.3333, A 0.000, B 0.000, C 0.000 }
gfCNCPoint1[7135] = {X 423.8886, Y 58.1782, Z -1.3333, A 0.000, B 0.000, C 0.000 }
gfCNCPoint1[7136] = {X 429.6420, Y 60.4207, Z -1.3333, A 0.000, B 0.000, C 0.000 }
gfCNCPoint1[7137] = {X 457.7814, Y 71.5847, Z -1.3333, A 0.000, B 0.000, C 0.000 }
gfCNCPoint1[7138] = {X 457.7801, Y 63.2813, Z -1.3333, A 0.000, B 0.000, C 0.000 }
gfCNCPoint1[7139] = {X 456.9207, Y 63.0562, Z -1.3333, A 0.000, B 0.000, C 0.000 }
gfCNCPoint1[7140] = {X 456.1240, Y 62.6630, Z -1.3333, A 0.000, B 0.000, C 0.000 }
gfCNCPoint1[7141] = {X 455.4226, Y 62.1179, Z -1.3333, A 0.000, B 0.000, C 0.000 }
gfCNCPoint1[7142] = {X 454.8450, Y 61.4429, Z -1.3333, A 0.000, B 0.000, C 0.000 }
gfCNCPoint1[7143] = {X 454.4147, Y 60.6657, Z -1.3333, A 0.000, B 0.000, C 0.000 }
gfCNCPoint1[7144] = {X 454.1493, Y 59.8179, Z -1.3333, A 0.000, B 0.000, C 0.000 }
gfCNCPoint1[7145] = {X 454.0596, Y 58.9340, Z -1.3333, A 0.000, B 0.000, C 0.000 }
gfCNCPoint1[7146] = {X 454.0596, Y 58.0000, Z -1.3333, A 0.000, B 0.000, C 0.000 }
gfCNCPoint1[7147] = {X 454.1699, Y 57.0209, Z -1.3333, A 0.000, B 0.000, C 0.000 }
gfCNCPoint1[7148] = {X 454.4953, Y 56.0909, Z -1.3333, A 0.000, B 0.000, C 0.000 }
gfCNCPoint1[7149] = {X 455.0195, Y 55.2566, Z -1.3333, A 0.000, B 0.000, C 0.000 }
gfCNCPoint1[7150] = {X 455.7162, Y 54.5599, Z -1.3333, A 0.000, B 0.000, C 0.000 }
gfCNCPoint1[7151] = {X 456.5505, Y 54.0357, Z -1.3333, A 0.000, B 0.000, C 0.000 }
gfCNCPoint1[7152] = {X 457.4805, Y 53.7103, Z -1.3333, A 0.000, B 0.000, C 0.000 }
gfCNCPoint1[7153] = {X 458.4596, Y 53.6000, Z -1.3333, A 0.000, B 0.000, C 0.000 }
gfCNCPoint1[7154] = {X 475.0000, Y 53.6000, Z -1.3333, A 0.000, B 0.000, C 0.000 }
gfCNCPoint1[7155] = {X 475.9791, Y 53.7103, Z -1.3333, A 0.000, B 0.000, C 0.000 }
gfCNCPoint1[7156] = {X 476.9091, Y 54.0357, Z -1.3333, A 0.000, B 0.000, C 0.000 }
gfCNCPoint1[7157] = {X 477.7434, Y 54.5599, Z -1.3333, A 0.000, B 0.000, C 0.000 }
gfCNCPoint1[7158] = {X 478.4401, Y 55.2566, Z -1.3333, A 0.000, B 0.000, C 0.000 }
gfCNCPoint1[7159] = {X 478.9643, Y 56.0909, Z -1.3333, A 0.000, B 0.000, C 0.000 }
gfCNCPoint1[7160] = {X 479.2897, Y 57.0209, Z -1.3333, A 0.000, B 0.000, C 0.000 }
gfCNCPoint1[7161] = {X 479.4000, Y 58.0000, Z -1.3333, A 0.000, B 0.000, C 0.000 }
gfCNCPoint1[7162] = {X 479.3998, Y 58.9704, Z -1.3333, A 0.000, B 0.000, C 0.000 }
gfCNCPoint1[7163] = {X 479.3039, Y 59.8484, Z -1.3333, A 0.000, B 0.000, C 0.000 }
gfCNCPoint1[7164] = {X 479.0346, Y 60.6896, Z -1.3333, A 0.000, B 0.000, C 0.000 }
gfCNCPoint1[7165] = {X 478.6027, Y 61.4601, Z -1.3333, A 0.000, B 0.000, C 0.000 }
gfCNCPoint1[7166] = {X 478.0256, Y 62.1287, Z -1.3333, A 0.000, B 0.000, C 0.000 }
gfCNCPoint1[7167] = {X 477.3266, Y 62.6686, Z -1.3333, A 0.000, B 0.000, C 0.000 }
gfCNCPoint1[7168] = {X 476.5338, Y 63.0581, Z -1.3333, A 0.000, B 0.000, C 0.000 }
gfCNCPoint1[7169] = {X 475.6792, Y 63.2813, Z -1.3333, A 0.000, B 0.000, C 0.000 }
gfCNCPoint1[7170] = {X 475.6796, Y 92.7052, Z -1.3333, A 0.000, B 0.000, C 0.000 }
gfCNCPoint1[7171] = {X 476.0479, Y 92.7997, Z -1.3333, A 0.000, B 0.000, C 0.000 }
gfCNCPoint1[7172] = {X 476.4112, Y 92.9115, Z -1.3333, A 0.000, B 0.000, C 0.000 }
gfCNCPoint1[7173] = {X 477.2384, Y 93.2872, Z -1.3333, A 0.000, B 0.000, C 0.000 }
gfCNCPoint1[7174] = {X 477.9702, Y 93.8257, Z -1.3333, A 0.000, B 0.000, C 0.000 }
gfCNCPoint1[7175] = {X 478.5750, Y 94.5038, Z -1.3333, A 0.000, B 0.000, C 0.000 }
gfCNCPoint1[7176] = {X 479.0266, Y 95.2922, Z -1.3333, A 0.000, B 0.000, C 0.000 }
gfCNCPoint1[7177] = {X 479.3056, Y 96.1569, Z -1.3333, A 0.000, B 0.000, C 0.000 }
gfCNCPoint1[7178] = {X 479.4000, Y 97.0605, Z -1.3333, A 0.000, B 0.000, C 0.000 }
gfCNCPoint1[7179] = {X 479.4000, Y 97.6949, Z -1.3333, A 0.000, B 0.000, C 0.000 }
gfCNCPoint1[7180] = {X 479.8800, Y 97.6949, Z -1.3333, A 0.000, B 0.000, C 0.000 }
gfCNCPoint1[7181] = {X 507.6820, Y 97.6949, Z -1.3333, A 0.000, B 0.000, C 0.000 }
gfCNCPoint1[7182] = {X 507.6820, Y 100.0949, Z -1.3333, A 0.000, B 0.000, C 0.000 }
gfCNCPoint1[7183] = {X 600.0148, Y 100.0949, Z -1.3333, A 0.000, B 0.000, C 0.000 }
gfCNCPoint1[7184] = {X 600.0671, Y 100.0697, Z -1.3333, A 0.000, B 0.000, C 0.000 }
gfCNCPoint1[7185] = {X 600.0947, Y 100.0187, Z -1.3333, A 0.000, B 0.000, C 0.000 }
gfCNCPoint1[7186] = {X 600.0965, Y 99.1431, Z -1.3333, A 0.000, B 0.000, C 0.000 }
gfCNCPoint1[7187] = {X 600.0965, Y 49.8790, Z -1.3333, A 0.000, B 0.000, C 0.000 }
gfCNCPoint1[7188] = {X 601.1110, Y 49.7518, Z -1.3333, A 0.000, B 0.000, C 0.000 }
gfCNCPoint1[7189] = {X 602.0768, Y 49.4160, Z -1.3333, A 0.000, B 0.000, C 0.000 }
gfCNCPoint1[7190] = {X 602.9514, Y 48.8863, Z -1.3333, A 0.000, B 0.000, C 0.000 }
gfCNCPoint1[7191] = {X 603.6965, Y 48.1860, Z -1.3333, A 0.000, B 0.000, C 0.000 }
gfCNCPoint1[7192] = {X 603.6965, Y 47.3867, Z -1.3333, A 0.000, B 0.000, C 0.000 }
gfCNCPoint1[7193] = {X 603.1502, Y 48.0719, Z -1.3333, A 0.000, B 0.000, C 0.000 }
gfCNCPoint1[7194] = {X 602.4789, Y 48.6352, Z -1.3333, A 0.000, B 0.000, C 0.000 }
gfCNCPoint1[7195] = {X 601.7093, Y 49.0544, Z -1.3333, A 0.000, B 0.000, C 0.000 }
gfCNCPoint1[7196] = {X 600.8720, Y 49.3127, Z -1.3333, A 0.000, B 0.000, C 0.000 }
gfCNCPoint1[7197] = {X 600.0000, Y 49.4000, Z -1.3333, A 0.000, B 0.000, C 0.000 }
gfCNCPoint1[7198] = {X 593.5565, Y 49.4000, Z -1.3333, A 0.000, B 0.000, C 0.000 }
gfCNCPoint1[7199] = {X 592.5988, Y 49.2945, Z -1.3333, A 0.000, B 0.000, C 0.000 }
gfCNCPoint1[7200] = {X 591.6870, Y 48.9831, Z -1.3333, A 0.000, B 0.000, C 0.000 }
gfCNCPoint1[7201] = {X 590.8648, Y 48.4806, Z -1.3333, A 0.000, B 0.000, C 0.000 }
gfCNCPoint1[7202] = {X 590.1717, Y 47.8112, Z -1.3333, A 0.000, B 0.000, C 0.000 }
gfCNCPoint1[7203] = {X 589.6410, Y 47.0071, Z -1.3333, A 0.000, B 0.000, C 0.000 }
gfCNCPoint1[7204] = {X 589.3741, Y 46.3664, Z -1.3333, A 0.000, B 0.000, C 0.000 }
gfCNCPoint1[7205] = {X 589.2113, Y 45.6918, Z -1.3333, A 0.000, B 0.000, C 0.000 }
gfCNCPoint1[7206] = {X 589.1565, Y 45.0000, Z -1.3333, A 0.000, B 0.000, C 0.000 }
gfCNCPoint1[7207] = {X 589.1565, Y 44.0638, Z -1.3333, A 0.000, B 0.000, C 0.000 }
gfCNCPoint1[7208] = {X 589.2615, Y 43.1277, Z -1.3333, A 0.000, B 0.000, C 0.000 }
gfCNCPoint1[7209] = {X 589.5614, Y 42.2346, Z -1.3333, A 0.000, B 0.000, C 0.000 }
gfCNCPoint1[7210] = {X 590.0428, Y 41.4249, Z -1.3333, A 0.000, B 0.000, C 0.000 }
gfCNCPoint1[7211] = {X 590.6839, Y 40.7347, Z -1.3333, A 0.000, B 0.000, C 0.000 }
gfCNCPoint1[7212] = {X 590.6854, Y 40.3069, Z -1.3333, A 0.000, B 0.000, C 0.000 }
gfCNCPoint1[7213] = {X 590.6843, Y 35.2156, Z -1.3333, A 0.000, B 0.000, C 0.000 }
gfCNCPoint1[7214] = {X 590.6841, Y 33.9382, Z -1.3333, A 0.000, B 0.000, C 0.000 }
gfCNCPoint1[7215] = {X 585.5192, Y 46.6830, Z -1.3333, A 0.000, B 0.000, C 0.000 }
gfCNCPoint1[7216] = {X 585.4476, Y 46.8466, Z -1.3333, A 0.000, B 0.000, C 0.000 }
gfCNCPoint1[7217] = {X 585.3694, Y 47.0071, Z -1.3333, A 0.000, B 0.000, C 0.000 }
gfCNCPoint1[7218] = {X 584.8417, Y 47.8075, Z -1.3333, A 0.000, B 0.000, C 0.000 }
gfCNCPoint1[7219] = {X 584.1532, Y 48.4747, Z -1.3333, A 0.000, B 0.000, C 0.000 }
gfCNCPoint1[7220] = {X 583.3365, Y 48.9769, Z -1.3333, A 0.000, B 0.000, C 0.000 }
gfCNCPoint1[7221] = {X 582.4111, Y 49.2946, Z -1.3333, A 0.000, B 0.000, C 0.000 }
gfCNCPoint1[7222] = {X 581.4384, Y 49.4000, Z -1.3333, A 0.000, B 0.000, C 0.000 }
gfCNCPoint1[7223] = {X 580.4664, Y 49.2878, Z -1.3333, A 0.000, B 0.000, C 0.000 }
gfCNCPoint1[7224] = {X 579.5433, Y 48.9635, Z -1.3333, A 0.000, B 0.000, C 0.000 }
gfCNCPoint1[7225] = {X 578.7146, Y 48.4433, Z -1.3333, A 0.000, B 0.000, C 0.000 }
gfCNCPoint1[7226] = {X 578.0214, Y 47.7529, Z -1.3333, A 0.000, B 0.000, C 0.000 }
gfCNCPoint1[7227] = {X 577.4979, Y 46.9263, Z -1.3333, A 0.000, B 0.000, C 0.000 }
gfCNCPoint1[7228] = {X 577.4375, Y 46.7968, Z -1.3333, A 0.000, B 0.000, C 0.000 }
gfCNCPoint1[7229] = {X 577.3813, Y 46.6655, Z -1.3333, A 0.000, B 0.000, C 0.000 }
gfCNCPoint1[7230] = {X 572.0976, Y 33.7454, Z -1.3333, A 0.000, B 0.000, C 0.000 }
gfCNCPoint1[7231] = {X 572.0980, Y 40.7321, Z -1.3333, A 0.000, B 0.000, C 0.000 }
gfCNCPoint1[7232] = {X 572.7430, Y 41.4213, Z -1.3333, A 0.000, B 0.000, C 0.000 }
gfCNCPoint1[7233] = {X 573.2261, Y 42.2322, Z -1.3333, A 0.000, B 0.000, C 0.000 }
gfCNCPoint1[7234] = {X 573.5252, Y 43.1275, Z -1.3333, A 0.000, B 0.000, C 0.000 }
gfCNCPoint1[7235] = {X 573.6264, Y 44.0660, Z -1.3333, A 0.000, B 0.000, C 0.000 }
gfCNCPoint1[7236] = {X 573.6264, Y 45.0000, Z -1.3333, A 0.000, B 0.000, C 0.000 }
gfCNCPoint1[7237] = {X 573.5140, Y 45.9884, Z -1.3333, A 0.000, B 0.000, C 0.000 }
gfCNCPoint1[7238] = {X 573.1824, Y 46.9263, Z -1.3333, A 0.000, B 0.000, C 0.000 }
gfCNCPoint1[7239] = {X 572.6569, Y 47.7553, Z -1.3333, A 0.000, B 0.000, C 0.000 }
gfCNCPoint1[7240] = {X 571.9608, Y 48.4472, Z -1.3333, A 0.000, B 0.000, C 0.000 }
gfCNCPoint1[7241] = {X 571.1286, Y 48.9676, Z -1.3333, A 0.000, B 0.000, C 0.000 }
gfCNCPoint1[7242] = {X 570.2018, Y 49.2905, Z -1.3333, A 0.000, B 0.000, C 0.000 }
gfCNCPoint1[7243] = {X 569.2264, Y 49.4000, Z -1.3333, A 0.000, B 0.000, C 0.000 }
gfCNCPoint1[7244] = {X 562.4443, Y 49.4000, Z -1.3333, A 0.000, B 0.000, C 0.000 }
gfCNCPoint1[7245] = {X 561.4652, Y 49.2897, Z -1.3333, A 0.000, B 0.000, C 0.000 }
gfCNCPoint1[7246] = {X 560.5352, Y 48.9643, Z -1.3333, A 0.000, B 0.000, C 0.000 }
gfCNCPoint1[7247] = {X 559.7009, Y 48.4401, Z -1.3333, A 0.000, B 0.000, C 0.000 }
gfCNCPoint1[7248] = {X 559.0042, Y 47.7434, Z -1.3333, A 0.000, B 0.000, C 0.000 }
gfCNCPoint1[7249] = {X 558.4800, Y 46.9091, Z -1.3333, A 0.000, B 0.000, C 0.000 }
gfCNCPoint1[7250] = {X 558.1546, Y 45.9791, Z -1.3333, A 0.000, B 0.000, C 0.000 }
gfCNCPoint1[7251] = {X 558.0443, Y 45.0000, Z -1.3333, A 0.000, B 0.000, C 0.000 }
gfCNCPoint1[7252] = {X 558.0443, Y 44.0640, Z -1.3333, A 0.000, B 0.000, C 0.000 }
gfCNCPoint1[7253] = {X 558.1491, Y 43.1276, Z -1.3333, A 0.000, B 0.000, C 0.000 }
gfCNCPoint1[7254] = {X 558.4492, Y 42.2343, Z -1.3333, A 0.000, B 0.000, C 0.000 }
gfCNCPoint1[7255] = {X 558.9310, Y 41.4246, Z -1.3333, A 0.000, B 0.000, C 0.000 }
gfCNCPoint1[7256] = {X 559.5730, Y 40.7348, Z -1.3333, A 0.000, B 0.000, C 0.000 }
gfCNCPoint1[7257] = {X 559.5730, Y 9.2681, Z -1.3333, A 0.000, B 0.000, C 0.000 }
gfCNCPoint1[7258] = {X 558.9279, Y 8.5788, Z -1.3333, A 0.000, B 0.000, C 0.000 }
